// TwinCAT 3 PLC project ExamplePlc
// Company: Sensata Technologies Mechanization
// ProgramVersion: 3.1.4023.0
// libraries:
//   Sensata_Common, * (Sensata Technologies)
//   Sensata_Data, * (Sensata Technologies)
//   Sensata_Device_Comm, * (Sensata Technologies)
//   Sensata_Laser, * (Sensata Technologies)
//   Sensata_Utilities, * (Sensata Technologies)
//   Tc2_Standard, * (Beckhoff Automation GmbH)
//   Tc2_System, * (Beckhoff Automation GmbH)
//   Tc2_Utilities, * (Beckhoff Automation GmbH)
//   Tc3_Module, * (Beckhoff Automation GmbH)
// project tree:
//   0 Program/ GVL_DataTransfer.TcGVL, GVL_HMITags.TcGVL, GVL_LaserMarkingParams.TcGVL, GVL_MESData.TcGVL, GVL_MESData_ActuatorAssembly.TcGVL, GVL_PriorOp.TcGVL, GVL_ProductLimits.TcGVL, GVL_Test.TcGVL, PRG_Main.TcPOU
//   1 Module/0 Machines/ FB_ExampleMachine.TcPOU
//   1 Module/1 Stations/ FB_ExampleStation.TcPOU
//   1 Module/2 Devices/ FB_ExampleDevice.TcPOU
//   / TMethodNames_Cohap.TcDUT, TASK_Main.TcTTO (not stored), TMethod_Controls.TcDUT
// real-time tasks:
//   TASK TASK_Main: cycle T#10ms, priority 20, ADS port 350

// ---- TMethodNames_Cohap.TcDUT
TYPE TMethodNames_Cohap :
STRUCT
	M_init : STRING := 'init';
	M_GetAsicandChannelCardVersion : STRING := 'getSICAndChannelCardVersions';
	M_GetDLLVersion : STRING := 'getDLLVersions';
	M_TestDummy : STRING := 'TestDummy';
	M_TestDummy2 : STRING := 'TestDummy2';
	M_PowerUp : STRING := 'PowerUp';
	M_PowerDown : STRING := 'PowerDown';
	M_readSerialNumber : STRING := 'readSerialNumber';
	M_ReadDeviceOutput : STRING := 'ReadDeviceOutput';
	M_ReadFastChannelData : STRING := 'SENT_readFastChannelData';
	M_initDUT : STRING := 'initDUT';
	M_initialize : STRING := 'initialize';
	
	M_InitLot : STRING := 'InitLot';
//	M_T1Step1 : STRING := '';
//	stM_InitLot	: STRING := 'InitLot';
	stM_t1Precal : STRING := 't1Precal';
	stM_t1Step2 : STRING := 't1Step2';
	stM_t1Step3 : STRING := 't1Step3';
	stM_t2Step1 : STRING := 't2Step1';
	stM_t2Step2 : STRING := 't2Step2';
	stM_t2Step3 : STRING := 't2Step3';	
END_STRUCT
END_TYPE

// ---- TMethod_Controls.TcDUT
TYPE TMethod_Controls :
STRUCT
//		bRunImpMethods_Trigger : BOOL;
//		bRunImpMethods_Result : BOOL;
		bInitializeDeviceComm_Trigger : BOOL;
		bInitializeDeviceComm_Result : BOOL;
		bSetCurrentDevice_Trigger : BOOL;
		bSetCurrentDevice_Result : BOOL;
		M_init_Trigger : BOOL;
        M_init_Result : BOOL;
        M_GetAsicandChannelCardVersion_Trigger : BOOL;
        M_GetAsicandChannelCardVersion_Result : BOOL;
        M_GetDLLVersion_Trigger : BOOL;
        M_GetDLLVersion_Result : BOOL;
        M_TestDummy_Trigger : BOOL;
        M_TestDummy_Result : BOOL;
		M_TestDummy2_Trigger : BOOL;
        M_TestDummy2_Result : BOOL;
        M_PowerUp_Trigger : BOOL;
        M_PowerUp_Result : BOOL;
        M_PowerDown_Trigger : BOOL;
        M_PowerDown_Result : BOOL;
        M_readSerialNumber_Trigger : BOOL;
        M_readSerialNumber_Result : BOOL;
        M_ReadDeviceOutput_Trigger : BOOL;
        M_ReadDeviceOutput_Result : BOOL;
		M_ReadFastChannelData_Trigger : BOOL;
        M_ReadFastChannelData_Result : BOOL;
        M_initDUT_Trigger : BOOL;
        M_initDUT_Result : BOOL;
        M_initialize_Trigger : BOOL;
        M_initialize_Result : BOOL;
		M_initLot_Trigger : BOOL;
		M_initLot_Result : BOOL;
		
		M_t1PreCal_Trigger : BOOL;
		M_t1PreCal_Result : BOOL;
		M_t1Step2_Trigger : BOOL;
		M_t1Step2_Result : BOOL;
		M_t1Step3_Trigger : BOOL;
		M_t1Step3_Result : BOOL;
		M_t2Step1_Trigger : BOOL;
		M_t2Step1_Result : BOOL;
		M_t2Step2_Trigger : BOOL;
		M_t2Step2_Result : BOOL;
		M_t2Step3_Trigger : BOOL;
		M_t2Step3_Result : BOOL;
END_STRUCT
END_TYPE

// ---- 0 Program/GVL_DataTransfer.TcGVL
{attribute 'qualified_only'}
VAR_GLOBAL
//InsertLotHistory
	dintEquipment_Id : DINT;//int
	
	strLot_ID : STRING;//varchar
	strDeviceID :STRING := 'ZSE3230';//varchar
	strAsicType:UDINT := 43;//int
	
//	strTestTime_L1: STRING:='2023/01/27 10:12:11.000';//datetime
//	udintfixture_L1: UDINT:=1;//tinyint
//	bTestStatus_L1 : STRING:='Good';//varchar
//	udintErrorcode_L1 : UDINT:=0;//bigint
//	SerialNumber_L1:UDINT:=180000;//bigint
//	PressureOut_L1:REAL:=1688653;//float
//	TemperatureOut_L1:REAL:=4592369;//float
	
//	bTestStatus_L2 : STRING;//varchar
//	strTestTime_L2: STRING:='2023/01/25 10:12:11.000';//datetime
//	udintErrorcode_L2 : UDINT;
//	udintfixture_L2: UDINT;//tinyint
//	SerialNumber_L2:UDINT;
//	PressureOut_L2:REAL;
//	TemperatureOut_L2:REAL;
//	dintEquipment_Id : DINT;
	
//	strLot_ID : STRING;
//	strDeviceID :STRING;
//	strAsicType:UDINT;//int
	//****************************//
	
	
	strTestTime_L1: STRING;//datetime
	udintfixture_L1: UDINT;//tinyint
	bTestStatus_L1 : STRING:='Good';//varchar
	udintErrorcode_L1 : UDINT:=0;//bigint
	SerialNumber_L1:UDINT;//bigint
	PressureOut_L1:REAL;//float
	TemperatureOut_L1:REAL;//float
	FFTPriorOPstatus_L1: STRING;
	CalT1PriorOPstatus_L1:STRING;
	CalT2PriorOPstatus_L1:STRING;
	ErrorCode_L1:UDINT;
	
	bTestStatus_L2 : STRING;//varchar
	strTestTime_L2: STRING;//datetime
	udintErrorcode_L2 : UDINT;
	udintfixture_L2: UDINT;//tinyint
	SerialNumber_L2:UDINT;
	PressureOut_L2:REAL;
	TemperatureOut_L2:REAL;
	FFTPriorOPstatus_L2: STRING;
	CalT1PriorOPstatus_L2:STRING;
	CalT2PriorOPstatus_L2:STRING;
	ErrorCode_L2:UDINT;//01- prior Op, 02- Invalid SN, 03-Cohap Communication fail
	
	//prior OP 
	
	SerialNumber_temp:UDINT := 989;
	PriorOpTestmode: STRING := 'CalNoBlow';
	PriorOpTestStatus:STRING;
	priorOpResult: STRING;

END_VAR

// ---- 0 Program/GVL_HMITags.TcGVL
{attribute 'qualified_only'}
VAR_GLOBAL
	//machine status 
	//*******
	//Add this line of code to a Program : GVL_HMI.intMachine_State := GVL_Main.fbMachine.P_enumState;
	//*******
	intMachine_State :INT;
	
	// ---------------------------------------------------------------------------
	// Config Screen
	// ---------------------------------------------------------------------------		
	strEngineerPassword: T_MaxString;
	bEngineerAccessAllowed: BOOL;
	strEngineerSetPassword: T_MaxString := 'password';
	bEngineerLogout: BOOL;
	
	//machine overview
	intGood_Parts : INT;
	intBad_Parts : INT;
	intTotal_Parts: INT;
	rYield : REAL;
	dintEquipment_Id : DINT := 191135;
	strSoftware_Rev : STRING := '1.0.0';
	strHMI_Rev : STRING := '1.0';
	bStartBtn : BOOL;
	bStopBtn : BOOL;
	bResetBtn : BOOL;
	bClearBtn : BOOL;
	bUser_Active : BOOL;
	udintPromptMessage : UDINT;
	strUser_Prompt : T_MaxString;
	bLoadDirection: BOOL;
	bDirectionIndicator: BOOL;
	bUserRetryBtn : BOOL;
	bUserAbortBtn : BOOL;
	intStationStatus: INT;
	
	bSetPartIdExternal : BOOL;
	bSetJobIdExternal : BOOL;
	bSetLotIdExternal : BOOL;
	
	strExternalPartId : STRING;
	strExternalJobId : STRING;
	strExternalLotId : STRING;
			
	//Lot Control
	bStart_Lot :BOOL;
	bEnd_Lot : BOOL;
	bLot_Active :BOOL;
	strLot_Num : STRING;
	strJob_Num : STRING;
	strPart_Num : STRING;
	bLimits_Loaded : Bool;
	
	//load unload
	strL1_HCode_Unload : STRING;
	strL2_HCode_Unload : STRING;
	strR1_HCode_Unload : STRING;
	strR2_HCode_Unload : STRING;
	bL1_State_Unload : BOOL;
	bL2_State_Unload : BOOL;
	bR1_State_Unload : BOOL;
	bR2_State_Unload : BOOL;
	
	//conditioner
	intNum_Cycles : INT;
	intOn_Time : INT;
	intOff_Time : INT;
	intCycles_Run :INT;
	bL1_Cond_State : BOOL;
	bL2_Cond_State : BOOL;
	bR1_Cond_State : BOOL;
	bR2_Cond_State : BOOL;
	strL1_Cond_HCode : STRING;
	strL2_Cond_HCode : STRING;
	strR1_Cond_HCode : STRING;
	strR2_Cond_HCode : STRING;
		
	//contact resistance	
	strCR_L1_HCode : STRING;
	rCR_L1_CR : REAL;
	rCR_L1_M1R : REAL;
	rCR_L1_M1V : REAL;
	rCR_L1_M1C : REAL;
	rCR_L1_M2R : REAL;
	rCR_L1_M2V : REAL;
	rCR_L1_M2C : REAL;
	rCR_L1_A1R : REAL;
	rCR_L1_A1V : REAL;
	rCR_L1_A1C : REAL;
	rCR_L1_A2R : REAL;
	rCR_L1_A2V : REAL;
	rCR_L1_A2C : REAL;
	bL1_CR_State : BOOL;
	
	strCR_L2_HCode : STRING;
	rCR_L2_CR : REAL;
	rCR_L2_M1R : REAL;
	rCR_L2_M1V : REAL;
	rCR_L2_M1C : REAL;
	rCR_L2_M2R : REAL;
	rCR_L2_M2V : REAL;
	rCR_L2_M2C : REAL;
	rCR_L2_A1R : REAL;
	rCR_L2_A1V : REAL;
	rCR_L2_A1C : REAL;
	rCR_L2_A2R : REAL;
	rCR_L2_A2V : REAL;
	rCR_L2_A2C : REAL;
	bL2_CR_State : BOOL;
	
	strCR_R1_HCode : STRING;
	rCR_R1_CR : REAL;
	rCR_R1_M1R : REAL;
	rCR_R1_M1V : REAL;
	rCR_R1_M1C : REAL;
	rCR_R1_M2R : REAL;
	rCR_R1_M2V : REAL;
	rCR_R1_M2C : REAL;
	rCR_R1_A1R : REAL;
	rCR_R1_A1V : REAL;
	rCR_R1_A1C : REAL;
	rCR_R1_A2R : REAL;
	rCR_R1_A2V : REAL;
	rCR_R1_A2C : REAL;	
	bR1_CR_State : BOOL;
	
	strCR_R2_HCode : STRING;
	rCR_R2_CR : REAL;
	rCR_R2_M1R : REAL;
	rCR_R2_M1V : REAL;
	rCR_R2_M1C : REAL;
	rCR_R2_M2R : REAL;
	rCR_R2_M2V : REAL;
	rCR_R2_M2C : REAL;
	rCR_R2_A1R : REAL;
	rCR_R2_A1V : REAL;
	rCR_R2_A1C : REAL;
	rCR_R2_A2R : REAL;
	rCR_R2_A2V : REAL;
	rCR_R2_A2C : REAL;
	bR2_CR_State : BOOL;
		
	//hipot	
	strHp_L1_HCode : STRING;
	strHp_L2_HCode : STRING;
	strHp_R1_HCode : STRING;
	strHp_R2_HCode : STRING;
	//to be deleted
	bL1_Hp_State : BOOL;
	bL2_Hp_State : BOOL;
	bR1_Hp_State : BOOL;	
	bR2_Hp_State : BOOL;
	
	rHp_FT_L1 : REAL;
	rHp_FT_L2 : REAL;
	rHp_FT_R1 : REAL;
	rHp_FT_R2 : REAL;

	rHp_Res_L1 : REAL;
	rHp_Res_L2 : REAL;
	rHp_Res_R1 : REAL;
	rHp_Res_R2 : REAL;
	
	strHp_Msg_L1 : STRING;
	strHp_Msg_L2 : STRING;
	strHp_Msg_R1 : STRING;
	strHp_Msg_R2 : STRING;
	
	HP_testName : STRING;
	//not used on HMI
	rHp_BDC_L1 : REAL;
	rHp_ARC_L1 : REAL;
	rHp_Result_L1 : REAL;
	rHp_BDC_L2 : REAL;
	rHp_ARC_L2 : REAL;
	rHp_Result_L2 : REAL;
	rHp_BDC_R1 : REAL;
	rHp_ARC_R1 : REAL;
	rHp_Result_R1 : REAL;
	rHp_BDC_R2 : REAL;
	rHp_ARC_R2 : REAL;
	rHp_Result_R2 : REAL;
	//AB proposed new Tags
	strNestAErrorMsg:STRING;
	strNestBErrorMsg:STRING;
	strNestCErrorMsg:STRING;
	strNestDErrorMsg:STRING;
	
	rHPMeasured_MML1:REAL;
	rHPMeasured_MML2:REAL;
	rHPMeasured_MMR1:REAL;
	rHPMeasured_MMR2:REAL;
	
	rHPMeasured_MMIRL1:REAL;
	rHPMeasured_MMIRL2:REAL;
	rHPMeasured_MMIRR1:REAL;
	rHPMeasured_MMIRR2:REAL;
	
	rHPMeasured_AAL1:REAL;
	rHPMeasured_AAL2:REAL;
	rHPMeasured_AAR1:REAL;
	rHPMeasured_AAR2:REAL;
	
	rHPMeasured_AuxIRL1:REAL;
	rHPMeasured_AuxIRL2:REAL;
	rHPMeasured_AuxIRR1:REAL;
	rHPMeasured_AuxIRR2:REAL;
	
	rHPMeasured_MainCoilopenL1:REAL;
	rHPMeasured_MainCoilopenL2:REAL;
	rHPMeasured_MainCoilopenR1:REAL;
	rHPMeasured_MainCoilopenR2:REAL;
	
	rHPMeasured_MainCoilIRL1:REAL;
	rHPMeasured_MainCoilIRL2:REAL;
	rHPMeasured_MainCoilIRR1:REAL;
	rHPMeasured_MainCoilIRR2:REAL;
	
	rHPMeasured_MainCoilClosedL1:REAL;
	rHPMeasured_MainCoilClosedL2:REAL;
	rHPMeasured_MainCoilClosedR1:REAL;
	rHPMeasured_MainCoilClosedR2:REAL;
	
	
	//PUV_DOV
	strPUV_L1_HCode : STRING;
	strPUV_L2_HCode : STRING;
	strPUV_R1_HCode : STRING;
	strPUV_R2_HCode : STRING;
	
	bL1_puv_State : BOOL;
	bL2_puv_State : BOOL;
	bR1_puv_State : BOOL;
	bR2_puv_State : BOOL;
	
	rPuv_L1 : REAL;
	rDov_L1 : REAL;	
	rPuc_L1 : REAL;
	rDoc_L1 : REAL;
	rPuv_L2 : REAL;
	rDov_L2 : REAL;	
	rPuc_L2 : REAL;
	rDoc_L2 : REAL;
	rPuv_R1 : REAL;
	rDov_R1 : REAL;	
	rPuc_R1 : REAL;
	rDoc_R1 : REAL;
	rPuv_R2 : REAL;
	rDov_R2 : REAL;	
	rPuc_R2 : REAL;
	rDoc_R2 : REAL;
	
	arrCoilPUV: ARRAY[1..4] OF LREAL;
	arrCoilDOV: ARRAY[1..4] OF LREAL;
	arrCoilResistance: ARRAY[1..4] OF LREAL;
		
	//functional test	
	strFT_L1_HCode : STRING;
	strFT_L2_HCode : STRING;
	strFT_R1_HCode : STRING;
	strFT_R2_HCode : STRING;
	
	bL1_ft_State : BOOL;
	bL2_ft_State : BOOL;
	bR1_ft_State : BOOL;
	bR2_ft_State : BOOL;
	
	MainOperatTime_L1 : REAL;
	MainReleaseTime_L1 : REAL;	
	AuxOperateTime_L1 : REAL;
	AuxReleaseTime_L1 : REAL;
	RSim_L1 : REAL;
	MainOperatTime_L2 : REAL;
	MainReleaseTime_L2 : REAL;	
	AuxOperateTime_L2 : REAL;
	AuxReleaseTime_L2 : REAL;
	RSim_L2 : REAL;
	MainOperatTime_R1 : REAL;
	MainReleaseTime_R1 : REAL;	
	AuxOperateTime_R1 : REAL;
	AuxReleaseTime_R1 : REAL;
	RSim_R1 : REAL;
	MainOperatTime_R2 : REAL;
	MainReleaseTime_R2 : REAL;	
	AuxOperateTime_R2 : REAL;
	AuxReleaseTime_R2 : REAL;
	RSim_R2 : REAL;
	
	//laser mark	
	bLaser_Connected_State : BOOL;
	bLaser_Mark_Status : BOOL;
	bLaser_Mark_Status_L1 : BOOL; //Marking Status of Part in Nest L1
	bLaser_Mark_Status_L2 : BOOL; //Marking Status of Part in Nest L2
	bLaser_Mark_Status_R1 : BOOL; //Marking Status of Part in Nest R1
	bLaser_Mark_Status_R2 : BOOL; //Marking Status of Part in Nest R2
	
	//Station PBs
	bDialTableRetry: BOOL;
	bDialTableAbort: BOOL;
	bCondRetry : BOOL;
	bCondAbort : BOOL;
	bCRRetry : BOOL;
	bCRAbort : BOOL;
	bHPRetry : BOOL;
	bHPAbort : BOOL;
	bPUVRetry : BOOL;
	bPUVAbort : BOOL;
	bFTRetry : BOOL;
	bFTAbort : BOOL;
	bLaserRetry: BOOL;
	bLaserAbort: BOOL;
	
	//Station Messages
	strLoadUserMsg : T_MaxString;
	strCondUserMsg : T_MaxString;
	strCRUserMsg : T_MaxString;
	strHPUserMsg : T_MaxString;
	strPUVUserMsg : T_MaxString;
	strFTUserMsg : T_MaxString;
	
	//Disable stations from HMI
	bDisableDialTable : BOOL;
	bDisableLoadUnload : BOOL;
	bDisableConditioner : BOOL;
	bDisableCR : BOOL;
	bDisableHiPot : BOOL;
	bDisableLaserMark : BOOL;
	bDisablePUVDOV : BOOL;
	bDisableFunctionTest : BOOL;	
	
	udintDialTablePrompt: UDINT;
	udintLoadUnloadPrompt: UDINT;
	udintConditionerPrompt: UDINT;
	udintContactResistancePrompt: UDINT;
	udintHiPotPrompt: UDINT;
	udintLaserPrompt: UDINT;
	udintPUVDOVPrompt: UDINT;
	udintFunctionTestPrompt: UDINT;
	
	bDialTablePromptActive: BOOL;
	bLoadUnloadPromptActive: BOOL;
	bConditionerPromptActive: BOOL;
	bContactResistancePromptActive: BOOL;
	bHiPotPromptActive: BOOL;
	bLaserPromptActive: BOOL;
	bPUVDOVPromptActive: BOOL;
	bFunctionTestPromptActive: BOOL;
	
	udintDialTableFault: UDINT;
	udintLoadUnloadFault: UDINT;
	udintConditionerFault: UDINT;
	udintContactResistanceFault: UDINT;
	udintHiPotFault: UDINT;
	udintLaserFault: UDINT;
	udintPUVDOVFault: UDINT;
	udintFunctionTestFault: UDINT;
	
	bDialTableFaulted: BOOL;
	bLoadUnloadFaulted: BOOL;
	bConditionerFaulted: BOOL;
	bContactResistanceFaulted: BOOL;
	bHiPotFaulted: BOOL;
	bLaserFaulted: BOOL;
	bPUVDOVFaulted: BOOL;
	bFunctionTestFaulted: BOOL;

	
	intDialTableState: INT;
	intLoadUnloadState: INT;
	intConditionerState: INT;
	intContactResistanceState: INT;
	intHiPotState: INT;
	intLaserState: INT;
	intPUVDOVState: INT;
	intFunctionTestState: INT;
	
	//Station and Nest failed consecutively 3 times
	//intStationNumFailed: INT;
	//intNestNumFailed: INT;
	arrStationNestNumFailed: ARRAY[1..2] OF INT;
	
	//IO Screen
	arrDigitalInputs: ARRAY[1..32] OF BOOL;
	arrRemoteInputs: ARRAY[1..48] OF BOOL;
	arrIOLinkInputs: ARRAY[1..4] OF BOOL;
	arrDigitalOutputStatus: ARRAY[1..120] OF BOOL;
	arrRelayOutputStatus: ARRAY[1..4] OF BOOL;
	arrPneumaticOutputStatus: ARRAY[1..32] OF BOOL;
	arrGuardDoors: ARRAY[1..16] OF BOOL;
//	arrMultiTimestampInputs: ARRAY[1..8] OF ST_EL1258_Inputs_Channel;
	
END_VAR

// ---- 0 Program/GVL_LaserMarkingParams.TcGVL
{attribute 'qualified_only'}
VAR_GLOBAL
	strHousingCode_L1 : STRING;	

	strCustomerDeviceID_L1 : STRING;
	strBlock0_L1 : STRING;
	strBlock1_L1 : STRING;
	strBlock2_L1 : STRING;
	strBlock3_L1 : STRING;
	strBlock4_L1 : STRING;
	strBlock5_L1 : STRING;
	strBlock6_L1 : STRING;
	strBlock7_L1 : STRING;
	strBlock8_L1 : STRING;
	strBlock9_L1 : STRING;
	strBlock10_L1 : STRING;
	
	strHousingCode_L2 : STRING;	
	
	strCustomerDeviceID_L2 : STRING;
	strBlock0_L2 : STRING;
	strBlock1_L2 : STRING;
	strBlock2_L2 : STRING;
	strBlock3_L2 : STRING;
	strBlock4_L2 : STRING;
	strBlock5_L2 : STRING;
	strBlock6_L2 : STRING;
	strBlock7_L2 : STRING;
	strBlock8_L2 : STRING;
	strBlock9_L2  : STRING;
	strBlock10_L2 : STRING;

	strHousingCode_R1 : STRING;	
	
	strCustomerDeviceID_R1 : STRING;
	strBlock0_R1 : STRING;
	strBlock1_R1 : STRING;
	strBlock2_R1 : STRING;
	strBlock3_R1 : STRING;
	strBlock4_R1 : STRING;
	strBlock5_R1 : STRING;
	strBlock6_R1 : STRING;
	strBlock7_R1 : STRING;
	strBlock8_R1 : STRING;
	strBlock9_R1 : STRING;
	strBlock10_R1 : STRING;
	
	strHousingCode_R2 : STRING;	
	
	strCustomerDeviceID_R2 : STRING;
	strBlock0_R2 : STRING;
	strBlock1_R2 : STRING;
	strBlock2_R2 : STRING;
	strBlock3_R2 : STRING;
	strBlock4_R2 : STRING;
	strBlock5_R2 : STRING;
	strBlock6_R2 : STRING;
	strBlock7_R2 : STRING;
	strBlock8_R2 : STRING;
	strBlock9_R2 : STRING;
	strBlock10_R2 : STRING;
	
END_VAR

// ---- 0 Program/GVL_MESData.TcGVL
{attribute 'qualified_only'}
VAR_GLOBAL
	//Lot Information
	LotBarcode : STRING;// := '80600600+57805702+23330166A+200';
	
	LotNo : STRING;
	ProductNo : STRING;
	OrderNo : STRING;
	Quantity : INT;
	OperatorID : STRING;
	ShiftLeader : STRING;
	MachineID : STRING;
	LotIdent : INT;
	PiecesLeft : INT;
	PiecesOK : INT;
	PiecesNOK : INT;
	LotInfoResponseMessages : ARRAY[1..100] OF STRING;
	
	//Operator Information 1
	OperatorBarcode : STRING;
	OperatorInfoResponse : STRING;	
	OperatorInfoResponseMessages : ARRAY[1..100] OF STRING;
	
	//Start Lot Information 1
	StartLotResponse : STRING;
	StartLotResponseMessages : ARRAY[1..100] OF STRING;
	
	//Prod Lot Components 1, 2 , 3
	Comp1_ident: LINT;          // Equivalent to private long ident;
   	Comp1_ident2: INT;          // Equivalent to private int ident2;
    Comp1_seria: STRING;        // Equivalent to private string seria;
    Comp1_quan: INT;            // Equivalent to private int quan;
    Comp1_result: INT;        // Equivalent to private short result;
    Comp1_resultText: STRING;   // Equivalent to private string resultText;
    Comp1_actualQuan: INT;      // Equivalent to private int actualQuan;
    Comp1_item: STRING;         // Equivalent to private string item;
	
	Comp2_ident: LINT;          // Equivalent to private long ident;
   	Comp2_ident2: INT;          // Equivalent to private int ident2;
    Comp2_seria: STRING;        // Equivalent to private string seria;
    Comp2_quan: INT;            // Equivalent to private int quan;
    Comp2_result: INT;        // Equivalent to private short result;
    Comp2_resultText: STRING;   // Equivalent to private string resultText;
    Comp2_actualQuan: INT;      // Equivalent to private int actualQuan;
    Comp2_item: STRING;         // Equivalent to private string item;
	
	Comp3_ident: LINT;          // Equivalent to private long ident;
   	Comp3_ident2: INT;          // Equivalent to private int ident2;
    Comp3_seria: STRING;        // Equivalent to private string seria;
    Comp3_quan: INT;            // Equivalent to private int quan;
    Comp3_result: INT;        // Equivalent to private short result;
    Comp3_resultText: STRING;   // Equivalent to private string resultText;
    Comp3_actualQuan: INT;      // Equivalent to private int actualQuan;
    Comp3_item: STRING;         // Equivalent to private string item;
	
	//ComponentsValidation 1, 2, 3
	ComponentValidation1Response : BOOL;
	ComponentValidation2Response : BOOL;
	ComponentValidation3Response : BOOL;
	
	//Get Machine Settings 1
	MachineSettingStructure : STRING;
	in_MachSetResult : BOOL;
	in_MachSetStructResponse : T_MaxString;
	
	//AddScrapCompByReason1
	
	//ScrapInfo
	ScrapCode : INT;
	ScrapCount : INT;
	ScrapCodeDescr : STRING;
	
	//Response 
	AddScrapComponentByReasonResponse : BOOL;
	
	//EndComponentLot1
	UsedComponentQuantity : INT;
	ComponentLotFinished : BOOL;
	//Response 
	EndLotComponentResponse : BOOL;
	
	
	//GetMachineDefects
	GetMachineDefects1Success : BOOL;
	Scrap1_ScrapCode : INT;
	Scrap1_ScrapCount : INT;
	Scrap1_ScrapCodeDescr : STRING;	
	
	//AddMESMachineEvent
	MESMachineID : STRING;
	MESStationID : INT;
	MESEventCode : STRING;
	MESEventMessage : STRING;
	MESEventType : INT;
	MESEventOperatorID : STRING;
	
	MESResponseEventID : LINT;
	
	//UpdateMESMachineEvent
	MESIsResolvedStatus : BOOL;
	MESResolutionNotes : STRING;
	MESDateTimeResolved : DATE;
	MESUpdateEventID : LINT;
	
END_VAR

// ---- 0 Program/GVL_MESData_ActuatorAssembly.TcGVL
{attribute 'qualified_only'}
VAR_GLOBAL
	//Lot Information
	LotBarcode : STRING;// := '80600600+57805702+23330166A+200';
	
	LotNo : STRING;
	ProductNo : STRING;
	OrderNo : STRING;
	Quantity : INT;
	OperatorID : STRING;
	ShiftLeader : STRING;
	MachineID : STRING;
	LotIdent : INT;
	PiecesLeft : INT;
	PiecesOK : INT;
	PiecesNOK : INT;
	LotInfoResponseMessages : ARRAY[1..100] OF STRING;
	
	//Operator Information 1
	OperatorBarcode : STRING;
	OperatorInfoResponse : STRING;	
	OperatorInfoResponseMessages : ARRAY[1..100] OF STRING;
	
	//machine settings
	
	//Start Lot Information 1
	StartLotResponse : STRING;
	StartLotResponseMessages : ARRAY[1..100] OF STRING;
	
	//Prod Lot Components 1, 2 , 3
	Comp1_ident: LINT;          // Equivalent to private long ident;
   	Comp1_ident2: INT;          // Equivalent to private int ident2;
    Comp1_seria: STRING;        // Equivalent to private string seria;
    Comp1_quan: INT;            // Equivalent to private int quan;
    Comp1_result: INT;        // Equivalent to private short result;
    Comp1_resultText: STRING;   // Equivalent to private string resultText;
    Comp1_actualQuan: INT;      // Equivalent to private int actualQuan;
    Comp1_item: STRING;         // Equivalent to private string item;
	
	Comp2_ident: LINT;          // Equivalent to private long ident;
   	Comp2_ident2: INT;          // Equivalent to private int ident2;
    Comp2_seria: STRING;        // Equivalent to private string seria;
    Comp2_quan: INT;            // Equivalent to private int quan;
    Comp2_result: INT;        // Equivalent to private short result;
    Comp2_resultText: STRING;   // Equivalent to private string resultText;
    Comp2_actualQuan: INT;      // Equivalent to private int actualQuan;
    Comp2_item: STRING;         // Equivalent to private string item;
	
	Comp3_ident: LINT;          // Equivalent to private long ident;
   	Comp3_ident2: INT;          // Equivalent to private int ident2;
    Comp3_seria: STRING;        // Equivalent to private string seria;
    Comp3_quan: INT;            // Equivalent to private int quan;
    Comp3_result: INT;        // Equivalent to private short result;
    Comp3_resultText: STRING;   // Equivalent to private string resultText;
    Comp3_actualQuan: INT;      // Equivalent to private int actualQuan;
    Comp3_item: STRING;         // Equivalent to private string item;
	
	//ComponentsValidation 1, 2, 3
	ComponentValidation1Response : BOOL;
	ComponentValidation2Response : BOOL;
	ComponentValidation3Response : BOOL;
	
	//Get Machine Settings 1
	MachineSettingStructure : STRING;
	in_MachSetResult : BOOL;
	in_MachSetStructResponse : T_MaxString;
	
	//AddScrapCompByReason1
	
	//ScrapInfo
	ScrapCode : INT;
	ScrapCount : INT;
	ScrapCodeDescr : STRING;
	
	//Response 
	AddScrapComponentByReasonResponse : BOOL;
	
	//EndComponentLot1
	UsedComponentQuantity : INT;
	ComponentLotFinished : BOOL;
	//Response 
	EndLotComponentResponse : BOOL;
	
	
	//GetMachineDefects
	GetMachineDefects1Success : BOOL;
	Scrap1_ScrapCode : INT;
	Scrap1_ScrapCount : INT;
	Scrap1_ScrapCodeDescr : STRING;	
	
	//AddMESMachineEvent
	MESMachineID : STRING;
	MESStationID : INT;
	MESEventCode : STRING;
	MESEventMessage : STRING;
	MESEventType : INT;
	MESEventOperatorID : STRING;
	
	MESResponseEventID : LINT;
	
	//UpdateMESMachineEvent
	MESIsResolvedStatus : BOOL;
	MESResolutionNotes : STRING;
	MESDateTimeResolved : DATE;
	MESUpdateEventID : LINT;
	
	
	
END_VAR

// ---- 0 Program/GVL_PriorOp.TcGVL
{attribute 'qualified_only'}
VAR_GLOBAL
	strHousingCode_L1 : STRING;
	bLaserMarked_L1 : BOOL;
END_VAR

// ---- 0 Program/GVL_ProductLimits.TcGVL
{attribute 'qualified_only'}
VAR_GLOBAL
	strPart_Num : STRING := 'GV354-006'; // := 'GXV600-009';
	strToolingBarcodeRequired : STRING;
	intBarcodeLocation : INT;
	
	
	//Conditioner Station
	bEnableConditioner : BOOL;
	intNumberOfCyclesToRun : INT := 500;
	intOperateTime : INT := 8;
	intReleaseTime : INT := 18;
	
	//CR Station
	bEnableCR : BOOL;
	bAuxPresent : BOOL;
	bEnableDipTest : BOOL;
	bEnableEMFTest : BOOL;
	bEndTestInRange : BOOL;
	intInitialWaitTime : INT;
	intMaxTestPulseTime : INT;
	intNumberofContResToCheck : INT;
	intNumberofPulses : INT;//Currently for rivian only
	intPulseOFFTime : INT;
	lrealInAuxResistanceMin : LREAL; 
	lrealInAuxResistanceMax : LREAL;
	lrealInCoilResistanceMin : LREAL; 
	lrealInCoilResistanceMax : LREAL; 
	lrealInMainsResistanceMin : LREAL;
	lrealInMainsResistanceMax : LREAL;
	lrealInMainsResistanceRangeMax : LREAL;
	lrealInMainsResistanceLastPointMax : LREAL;	
	lrealSetCurrentCoil : LREAL;
	lrealSetVoltageCoil : LREAL;
	lrealSetCloseTestCurrentMain : LREAL;
	lrealSetCloseTestVoltageMain : LREAL;
	lrealSetTestingCurrentMain : LREAL;
	lrealSetTestingVoltageMain : LREAL;
	lrealMainsCurrentErrorPct : LREAL;

	bEnableHP:BOOL;
	bDBParamsAux2APresent:BOOL:=TRUE;
	bDBParamsAux2BPresent:BOOL;
	udintEquipmentCountCycle:UDINT;
	lrealTestVoltageHP:LREAL;
	lrealDwellTime:LREAL;
	lrealRampTime:LREAL;
	lrealMinCurrentHP:LREAL;
	lrealMaxCurrentHP:LREAL;
	lrealTestVoltageIR:LREAL;
	lrealMinResistanceIR:LREAL;
	lrealMaxResistanceIR:LREAL;
	strDUT_HP:STRING;
	
	//TestVoltage for Aux test
	lrTestVoltageAuxHP: LREAL;
	//DwellTime for Aux-Aux HP test
	lrTestDwellTimeAuxHP:LREAL;
	//RampTime for Aux-Aux HP test
	lrTestRampTimeAuxHP :LREAL;
	//MinAcceptable current for Aux-Aux HP test
	lrMinCurrentAuxHP :LREAL;
	//MaxAcceptable current for Aux-Aux HP test
	lrMaxCurrentAuxHP :LREAL;
	
	//PUVDOV Station
	bEnablePUV:BOOL;
	bBinarySearchEnabled: BOOL; 	
	bVoltageTest: BOOL;        	
	udintBinarySearchPoints : UDINT;	
	timeContactCloseCheck : UINT; 	
	timePowerFailCheck: UINT;
	timePowerSupplyStabilize: UINT;	
	lrealDefaultErrValue : LREAL;
	lrealPickUpUSLVoltage: LREAL;	
	lrealPickUpLSLVoltage: LREAL; 
	lrealPickUpBufferVoltage: LREAL;
	lrealPickUpUSLCurrent: LREAL;
	lrealPickUpLSLCurrent: LREAL;
	lrealPickUpBufferCurrent: LREAL;
	lrealCoilNominalVoltage: LREAL; 
	lrealCoilNominalCurrent: LREAL;
	lrealDropOutUSLVoltage: LREAL; 
	lrealDropOutLSLVoltage: LREAL;
	lrealDropOutBufferVoltage: LREAL;	
	lrealDropOutUSLCurrent: LREAL;	
	lrealDropOutLSLCurrent: LREAL;
	lrealDropOutBufferCurrent: LREAL;
	lrealMaxCurrentSet: LREAL;
	lrealMaxVoltageSet: LREAL;
	
	//Laser Station
	bEnableLaser:BOOL;
	strLaserBlock_0:STRING;
	strLaserBlock_1:STRING;
	strLaserBlock_2:STRING;
	strLaserBlock_3:STRING;
	strLaserBlock_4:STRING;
	strLaserBlock_5:STRING;
	strLaserBlock_6:STRING;
	strLaserBlock_7:STRING;
	strLaserBlock_8:STRING;
	strLaserBlock_9:STRING;
	strLaserBlock_10:STRING;
	
	//FT Station
	bEnableFT:BOOL;
	realMainsOTMin : REAL;
	realMainsOTMax : REAL;
	realAuxOTMin : REAL;
	realAuxOTMax : REAL;
	realMainsRTMin : REAL;
	realMainsRTMax : REAL;
	realAuxRTMin : REAL;
	realAuxRTMax : REAL;
	realRSimMin :REAL;
	realRSimMax:REAL;
	
	//Tooling Barcode
	strExpectedToolingBarcode: Tc2_System.T_MaxString;//Remove after db update 
	
	//Pallet Barcode
	strExpectedPalletBarcode : Tc2_System.T_MaxString;
END_VAR

// ---- 0 Program/GVL_Test.TcGVL
{attribute 'qualified_only'}
VAR_GLOBAL
	temperature : REAL;
	Pressure : REAL;
	
	startCommand : BOOL;
	stopCommand : BOOL;
	
END_VAR

// ---- 0 Program/PRG_Main.TcPOU
PROGRAM PRG_Main
VAR
	bTestInput: BOOL;
	bTestOutput: BOOL;
	fbMachine: FB_ExampleMachine;
	fbStation1: FB_ExampleStation;
	fbStation2: FB_ExampleStation;
	fbStation3: FB_ExampleStation;
	fbStation4: FB_ExampleStation;
	bStart: BOOL;
	bAbort: BOOL;
	bReset: BOOL;
	bStop: BOOL;
	bSuspend: BOOL;
	fbDevice1: FB_ExampleDevice;
	fbDevice2: FB_ExampleDevice;
	fbDevice3: FB_ExampleDevice;
	fbDevice4: FB_ExampleDevice;
	bPoweredOn: BOOL;
//	FB_AdsDeviceAPI_0: FB_AdsDeviceAPI;
	FB_AdsDeviceAPI_0 : FB_AdsCommandRouter;
//	FB_AdsDeviceAPI_1 : FB_AdsCommandRouter;
	MyLaser1: FB_KeyenceLaserMarkerMDX2000;
	(* Database handler FB. *)
//	in_fbDataHandler: REFERENCE TO FB_Data;

///////////////////////////////////////////////////////////////////////////
///////////////Laser Marking Testing////////////////////////////////////
///////////////////////////////////////////////////////////////////////////


	bConnectToLaserMarker: BOOL;
	bRes_LaserConnected: BOOL;
	
	bTestADSServer: BOOL;
	strTarget: T_MaxString;
	strCommand: T_MaxString;
	arrParams: T_ApiMethodParameters;
	MyResults: T_MaxString;
	bInterfaceTest : BOOL;
	temp: BOOL;
	
	
	bDisconnectFromLaserMarker: BOOL;
	bRes_LaserDisconnected: BOOL;
	
	bPeakCurrentProgramInLaser: BOOL;
	bRes_PeakCurrentProgramInLaser: BOOL;
	
	bSendProgramToLaser: BOOL;
	bRes_SendProgramtoLaser: BOOL;
	filepath : STRING;
	LaserMemoryLocation : INT;
	
	bSaveCurrentLaserProgramtoPC : BOOL;
	bRes_SaveCurrentLaserProgramtoPC: BOOL;
	LaserProgramFolderPath: STRING;
	
	bGetCurrentProgram : BOOL;
	bRes_GetCurrentProgram : BOOL;
	CurrentProgramName : T_MaxString;
	
	bStartMarking: BOOL;
	bRes_StartMarking: BOOL;
	
	bStopMarking: BOOL;
	bRes_StopMarking: BOOL;
	
	bClearLaserErrors: BOOL;
	bRes_ClearLaserErrors: BOOL;
	
	bUpdateProgramBlockInTheLaser: BOOL;
	bRes_UpdateProgramBlockInTheLaser: BOOL;
	_blockNumber: INT;
	_blockData: STRING;
	_blockType : BlockTypes;
	
	bGetLaserStatus: BOOL;
	bRes_GetLaserStatus: BOOL;
	_string_laserstatus : STRING;
	
	bGetLaserErrorStatus: BOOL;
	bRes_GetLaserErrorStatus: BOOL;
	_bIsLaserError : BOOL;
	
	bGetLaserActivatedStatus: BOOL;
	bRes_GetLaserActivatedStatus: BOOL;
	_bIsLaserActivated : BOOL;
	
	bGetLaserMarkingStatus: BOOL;
	bRes_GetLaserMarkingStatus: BOOL;
	_bIsLaserMarking : BOOL;
	
	bRes_Reset: BOOL;
	bResetErrors: BOOL;
	
	bUpdateProgramBlockMarkEnabledInTheLaser: BOOL;
	bRes_UpdateProgramBlockMarkEnabledInTheLaser: BOOL;
	_bool_markenabled : BOOL;
	_blockType_enum : BlockTypes;
	
	UpdateSingleBlockMarkEnabledIntheLaser_Success: BOOL;
	_bUpdateSingleBlockDataSuccess : BOOL;
	_bUpdateSingleBlockMarkEnabled_Success : BOOL;
	
	bUpdateAllMarkingInfo: BOOL;
	LastBlockToMark : INT;
	_OneTimeArrayBuild : BOOL := TRUE;
	BlockInfoArray : ARRAY [0..255] OF OneBlockInfo;
	bRes_UpdateAllMarkingInfo: BOOL;
	
	
	intIndex: INT;
	intIndex2 : INT;
	inst_intStep: INT := 0;
	_tempString : STRING;
	
	bRes_UpdateAllMarkInfo : ARRAY [0..255] OF BOOL;
	bUpdateAllMarkingInfo_MethodCall: BOOL;
	bRes_UpdateAllMarkingInfo_MethodCall: BOOL;
	
	
	fbDataHandler: FB_DataTracker;
	fbDataHandler2: FB_DataTracker;
	fbDatabaseCommandRouter: FB_AdsCommandRouter;
	_inst_bDataTransferred: BOOL;
	
	// (* Name of the parameters database transfer ID. *)
	in_strParametersDatabaseName: T_MaxString := 'GetLimits';
	in_strParametersDBNameLaserLimits_L1 : T_MaxString := 'GetLaserMarkingParams_L1';
	in_strParametersDBNameLaserLimits_L2 : T_MaxString := 'GetLaserMarkingParams_L2';
	in_strParametersDBNameLaserLimits_R1 : T_MaxString := 'GetLaserMarkingParams_R1';
	in_strParametersDBNameLaserLimits_R2 : T_MaxString := 'GetLaserMarkingParams_R2';	
	_inst_bLaserLimitsDataTransferred_L1 : BOOL;
	_inst_bLaserLimitsDataTransferred_L2 : BOOL;
	_inst_bLaserLimitsDataTransferred_R1 : BOOL;
	_inst_bLaserLimitsDataTransferred_R2 : BOOL;
	
	bGetLimitsFromDB : BOOL;
	
	bGetLaserParamsFromDB_L1 : BOOL;
	bGetLaserParamsFromDB_L2 : BOOL;
	bGetLaserParamsFromDB_R1 : BOOL;
	bGetLaserParamsFromDB_R2 : BOOL;
	
	bPerformPriorOp_Smart: BOOL;
	in_strParametersDBName_SmartWater : T_MaxString := 'GetPriorOPA';
	_inst_bPriorOp_Smart: BOOL;
	
	bPerformPriorOp_FFT: BOOL;
	in_strParametersDBName_FFTLaser_L1 : T_MaxString := 'LaserMarkCheckL1';
	_inst_bPriorOp_FFT: BOOL;
	
	Temp_CR_LOOKUP_NestL1 : INT;
	iLengthDataMatrixNestL1 : INT;
	ParamsArrayNestA : STRING;
	
///////////////////////////////////////////////////////////////////////////
///////////////MES Data Tracking Testing////////////////////////////////////
///////////////////////////////////////////////////////////////////////////

	
	fbDataHandler3: FB_MESDataTracking;
	bPerformGetLotInfoFromLotBarcode: BOOL;
	_inst_bGetLotInfo_LotBarcode: BOOL;
	in_strParamDBName_GetLotInfo: T_MaxString := 'GetLotInfo1';
	
	bPerformGetOpInfoFromOpBarcode: BOOL;
	in_strParamDBName_GetOpInfo: T_MaxString := 'GetOperatorInfo1';
	_inst_bGetOpInfo_OpBarcode: BOOL;
	
	bPerformStartLot : BOOL;
	_inst_bStartLot : BOOL;
	in_strParamDBName_StartLot : T_MaxString := 'StartLot1';
	
	bPerformGetProdLotComponents : BOOL;
	_inst_bGetProdLotComponents : BOOL;
	in_strParamDBName_GetProdLotComps : T_MaxString := 'GetProdLotComponents1';
	
	bPerformComponentValidation1 : BOOL;
	_inst_bCompValidation1 : BOOL;
	in_strParamDBName_Comp1Validation1 : T_MaxString := 'ComponentValidation1';
	
	bPerformComponentValidation2 : BOOL;
	_inst_bCompValidation2 : BOOL;
	in_strParamDBName_Comp1Validation2 : T_MaxString := 'ComponentValidation2';
	
	bPerformComponentValidation3 : BOOL;
	_inst_bCompValidation3 : BOOL;
	in_strParamDBName_Comp1Validation3 : T_MaxString := 'ComponentValidation3';
	
	bPerformGetMachineSettings : BOOL;
	_inst_bGetMachineSettings : BOOL;
	in_strParamDBName_GetMachSetting : T_MaxString := 'GetMachineSettings1';
	
	bPerformAddScrapCompByReason : BOOL;
	_inst_bAddScrapCompByReason : BOOL;
	in_strParamDBName_AddScrapCompByReason : T_MaxString := 'AddScrapComponentByReason1';
	
	bPerformEndLotComp : BOOL;
	_inst_bEndLotComp : BOOL;
	in_strParamDBName_EndLotComp : T_MaxString := 'EndLotComponent1';
	
	bPerformGetMachineDefects : BOOL;
	_inst_bGetMachineDefects : BOOL;
	in_strParamDBName_GetMachDefects : T_MaxString := 'GetMachineDefects1';

	
///////////////////////////////////////////////////////////////////////////
/////////////Testing Cohap Related Vars////////////////////////////////////
///////////////////////////////////////////////////////////////////////////

	//Initialize Only	
	MyCohapTest : FB_COHAP;
	bInitializeCohapSystem: BOOL;
	bRes_CohapConnected: BOOL;

//	//Execute RunImpMethods Only	;
	bExecuteRunImpMethods: BOOL;
	bRes_RunImpMethods: BOOL;

//	//Set Current Device Instance
	bSetCurrentDevice_Cohap : BOOL;
	bRes_SetCurrentDevice : BOOL;
//	//Input Params
	strDeviceName : STRING;
	
	//RunCommand
	bRunCommandCohapSystem : BOOL;
	bRes_RunCommand : BOOL;
	
	//Input Params
	strMethodName : STRING;
	RunCom_InpuParams : T_CohapParameterList;
	RunCom_ExpOutParamList : ARRAY[0..9] OF ST_ReturnParamsInfo;
	
	//Output Params
	RunCom_OutputParams : T_CohapParameterList;
	
	//DummyTest Dictionary Prep for RunCommand Execution
	RC_DT_InpPar : T_CohapParameterList;
	RC_DT_ExpOutPL : ARRAY[0..9] OF ST_ReturnParamsInfo;
	
	CohapMethodStrings : TMethodNames_Cohap;
	CohapMethodControls : TMethod_Controls;
//	fbCohapHandler1: FB_COHAP;

///////////////////////////////

	// For readSerialNumber
	readSerialNumber_inpuparams : T_CohapParameterList;
	readSerialNumber_expoutparamlist : ARRAY[0..9] OF ST_ReturnParamsInfo;
	readSerialNumber_outputparams : T_CohapParameterList;
	
	// For ReadDeviceOutput
	ReadDeviceOutput_inpuparams : T_CohapParameterList;
	ReadDeviceOutput_expoutparamlist : ARRAY[0..9] OF ST_ReturnParamsInfo;
	ReadDeviceOutput_outputparams : T_CohapParameterList;

	
	// For PowerUp
	PowerUp_inpuparams : T_CohapParameterList;
	PowerUp_expoutparamlist : ARRAY[0..9] OF ST_ReturnParamsInfo;
	PowerUp_outputparams : T_CohapParameterList;
	
	// For PowerDown
	PowerDown_inpuparams : T_CohapParameterList;
	PowerDown_expoutparamlist : ARRAY[0..9] OF ST_ReturnParamsInfo;
	PowerDown_outputparams : T_CohapParameterList;
	
	// For TestDummy
	TestDummy_inpuparams : T_CohapParameterList;
	TestDummy_expoutparamlist : ARRAY[0..9] OF ST_ReturnParamsInfo;
	TestDummy_outputparams : T_CohapParameterList;
	
	// For TestDummy2
	TestDummy2_inpuparams : T_CohapParameterList;
	TestDummy2_expoutparamlist : ARRAY[0..9] OF ST_ReturnParamsInfo;
	TestDummy2_outputparams : T_CohapParameterList;
	
	// For init
	init_inpuparams : T_CohapParameterList;
	init_expoutparamlist : ARRAY[0..9] OF ST_ReturnParamsInfo;
	init_outputparams : T_CohapParameterList;
	
	// For getSICAndChannelCardVersions
	getSICAndChannelCardVersions_inpuparams : T_CohapParameterList;
	getSICAndChannelCardVersions_expoutparamlist : ARRAY[0..9] OF ST_ReturnParamsInfo;
	getSICAndChannelCardVersions_outputparams : T_CohapParameterList;
	
	// For getDLLVersions
	getDLLVersions_inpuparams : T_CohapParameterList;
	getDLLVersions_expoutparamlist : ARRAY[0..9] OF ST_ReturnParamsInfo;
	getDLLVersions_outputparams : T_CohapParameterList;
	
	// For initDUT
	initDUT_inpuparams : T_CohapParameterList;
	initDUT_expoutparamlist : ARRAY[0..9] OF ST_ReturnParamsInfo;
	initDUT_outputparams : T_CohapParameterList;
	
	//For Fast Channel Data
	readFastChannelData_inputparams : T_CohapParameterList;
	readFastChannelData_expoutparamlist : ARRAY[0..9] OF ST_ReturnParamsInfo;
	readFastChannelData_outputparams : T_CohapParameterList;

	// For T1 Step 1 Calibration
	t1Step1_inpuparams : T_CohapParameterList;
	t1Step1_expoutparamlist : ARRAY[0..9] OF ST_ReturnParamsInfo;
	t1Step1_outputparams : T_CohapParameterList;
	
//	// For T1 Step 2 Calibration
//	t1Step2_inpuparams : T_CohapParameterList;
//	t1Step2_expoutparamlist : ARRAY[0..9] OF ST_ReturnParamsInfo;
//	t1Step2_outputparams : T_CohapParameterList;
	
//	// For T1 Step 3 Calibration
//	t1Step3_inpuparams : T_CohapParameterList;
//	t1Step3_expoutparamlist : ARRAY[0..9] OF ST_ReturnParamsInfo;
//	t1Step3_outputparams : T_CohapParameterList;
	
	// For T2 Step 1 Calibration
	t2Step1_inpuparams : T_CohapParameterList;
	t2Step1_expoutparamlist : ARRAY[0..9] OF ST_ReturnParamsInfo;
	t2Step1_outputparams : T_CohapParameterList;
	
	// For T2 Step 2 Calibration
	t2Step2_inpuparams : T_CohapParameterList;
	t2Step2_expoutparamlist : ARRAY[0..9] OF ST_ReturnParamsInfo;
	t2Step2_outputparams : T_CohapParameterList;
	
	// For T2 Step 3 Calibration
	t2Step3_inpuparams : T_CohapParameterList;
	t2Step3_expoutparamlist : ARRAY[0..9] OF ST_ReturnParamsInfo;
	t2Step3_outputparams : T_CohapParameterList;
	
	// InitLot Device12133 class in Mech Device Lib Calibration
	InitLot_inputparams : T_CohapParameterList;
	InitLot_expoutparamlist : ARRAY[0..9] OF ST_ReturnParamsInfo;
	InitLot_outputparams : T_CohapParameterList;
	
//	//For Init Lot
//	InitLot_inputparams : T_CohapParameterList;
//	InitLot_expoutparamlist : ARRAY[0..9] OF ST_ReturnParamsInfo;
//	InitLot_outputparams : T_CohapParameterList;	
	// For T1 Step 1 Calibration
	t1Precal_inputparams : T_CohapParameterList;
	t1Precal_expoutparamlist : ARRAY[0..9] OF ST_ReturnParamsInfo;
	t1Precal_outputparams : T_CohapParameterList;
	// For T1 Step 2 Calibration
	t1Step2_inputparams : T_CohapParameterList;
	t1Step2_expoutparamlist : ARRAY[0..9] OF ST_ReturnParamsInfo;
	t1Step2_outputparams : T_CohapParameterList;
	// For T1 Step 3 Calibration
	t1Step3_inputparams : T_CohapParameterList;
	t1Step3_expoutparamlist : ARRAY[0..9] OF ST_ReturnParamsInfo;
	t1Step3_outputparams : T_CohapParameterList;
	
END_VAR
VAR // added by the converter: edge detectors and wires of the graphical bodies
    _w1, _w2, _w3, _w4, _w5, _w6, _w7, _w8, _w9, _w10, _w11, _w12, _w13, _w14, _w15, _w16, _w17, _w18, _w19, _w20, _w21, _w22, _w23, _w24, _w25, _w26, _w27, _w28, _w29, _w30, _w31, _w32, _w33, _w34, _w35, _w36, _w37, _w38, _w39, _w40 : BOOL;
END_VAR

bTestOutput := bTestInput;

A_Machine();
M_TestMESVars();
M_TestLaserMarker();
M_TestCohapLibrary();
//A_CohapLibraryTesting();
//A_InitCohapMethodParams();
//A_CohapLDTesting();

//A_Station1();
//A_Station2();
//A_Station3();
//A_Station4();
//bInterfaceTest := MyLaser1.fbApi.P_bDeviceInterfaceBusy;



//IF bPerformGetLotInfoFromLotBarcode THEN
//	_inst_bGetLotInfo_LotBarcode := fbDataHandler3.M_TransferData(in_strParamDBName_GetLotInfo);
//	IF _inst_bGetLotInfo_LotBarcode THEN
//		bPerformGetLotInfoFromLotBarcode := FALSE;
//	ELSIF fbDataHandler3.P_bError THEN 
//		bPerformGetLotInfoFromLotBarcode := FALSE;
//		fbDataHandler3.M_ClearError();
//	END_IF
//END_IF

//IF bPerformGetOpInfoFromOpBarcode THEN
//	_inst_bGetOpInfo_OpBarcode := fbDataHandler3.M_TransferData(in_strParamDBName_GetOpInfo);
//	IF _inst_bGetOpInfo_OpBarcode THEN
//		bPerformGetOpInfoFromOpBarcode := FALSE;
//	ELSIF fbDataHandler3.P_bError THEN 
//		bPerformGetOpInfoFromOpBarcode := FALSE;
//		fbDataHandler3.M_ClearError();
//	END_IF
//END_IF

//IF bPerformStartLot THEN
//	_inst_bStartLot := fbDataHandler3.M_TransferData(in_strParamDBName_StartLot);
//	IF _inst_bStartLot THEN
//		bPerformStartLot := FALSE;
//	ELSIF fbDataHandler3.P_bError THEN 
//		bPerformStartLot := FALSE;
//		fbDataHandler3.M_ClearError();
//	END_IF
//END_IF

//IF bPerformGetProdLotComponents THEN
//	_inst_bGetProdLotComponents := fbDataHandler3.M_TransferData(in_strParamDBName_GetProdLotComps);
//	IF _inst_bGetProdLotComponents THEN
//		bPerformGetProdLotComponents := FALSE;
//	ELSIF fbDataHandler3.P_bError THEN 
//		bPerformGetProdLotComponents := FALSE;
//		fbDataHandler3.M_ClearError();
//	END_IF
//END_IF


//IF bPerformComponentValidation1 THEN
//	_inst_bCompValidation1 := fbDataHandler3.M_TransferData(in_strParamDBName_Comp1Validation1);
//	IF _inst_bCompValidation1 THEN
//		bPerformComponentValidation1 := FALSE;
//	ELSIF fbDataHandler3.P_bError THEN 
//		bPerformComponentValidation1 := FALSE;
//		fbDataHandler3.M_ClearError();
//	END_IF
//END_IF

//IF bPerformComponentValidation2 THEN
//	_inst_bCompValidation2 := fbDataHandler3.M_TransferData(in_strParamDBName_Comp1Validation2);
//	IF _inst_bCompValidation2 THEN
//		bPerformComponentValidation2 := FALSE;
//	ELSIF fbDataHandler3.P_bError THEN 
//		bPerformComponentValidation2 := FALSE;
//		fbDataHandler3.M_ClearError();
//	END_IF
//END_IF

//IF bPerformComponentValidation3 THEN
//	_inst_bCompValidation3 := fbDataHandler3.M_TransferData(in_strParamDBName_Comp1Validation3);
//	IF _inst_bCompValidation3 THEN
//		bPerformComponentValidation3 := FALSE;
//	ELSIF fbDataHandler3.P_bError THEN 
//		bPerformComponentValidation3 := FALSE;
//		fbDataHandler3.M_ClearError();
//	END_IF
//END_IF

//IF bPerformGetMachineSettings THEN
//	_inst_bGetMachineSettings := fbDataHandler3.M_TransferData(in_strParamDBName_GetMachSetting);
//	IF _inst_bGetMachineSettings THEN
//		bPerformGetMachineSettings := FALSE;
//	ELSIF fbDataHandler3.P_bError THEN 
//		bPerformGetMachineSettings := FALSE;
//		fbDataHandler3.M_ClearError();
//	END_IF
//END_IF

//IF bPerformAddScrapCompByReason THEN
//	_inst_bAddScrapCompByReason := fbDataHandler3.M_TransferData(in_strParamDBName_AddScrapCompByReason);
//	IF _inst_bAddScrapCompByReason THEN
//		bPerformAddScrapCompByReason := FALSE;
//	ELSIF fbDataHandler3.P_bError THEN 
//		bPerformAddScrapCompByReason := FALSE;
//		fbDataHandler3.M_ClearError();
//	END_IF
//END_IF

//IF bPerformEndLotComp THEN
//	_inst_bEndLotComp := fbDataHandler3.M_TransferData(in_strParamDBName_EndLotComp);
//	IF _inst_bEndLotComp THEN
//		bPerformEndLotComp := FALSE;
//	ELSIF fbDataHandler3.P_bError THEN 
//		bPerformEndLotComp := FALSE;
//		fbDataHandler3.M_ClearError();
//	END_IF
//END_IF

//IF bPerformGetMachineDefects THEN
//	_inst_bGetMachineDefects := fbDataHandler3.M_TransferData(in_strParamDBName_GetMachDefects);
//	IF _inst_bGetMachineDefects THEN
//		bPerformGetMachineDefects := FALSE;
//	ELSIF fbDataHandler3.P_bError THEN 
//		bPerformGetMachineDefects := FALSE;
//		fbDataHandler3.M_ClearError();
//	END_IF
//END_IF

ACTION A_CohapLDTesting:
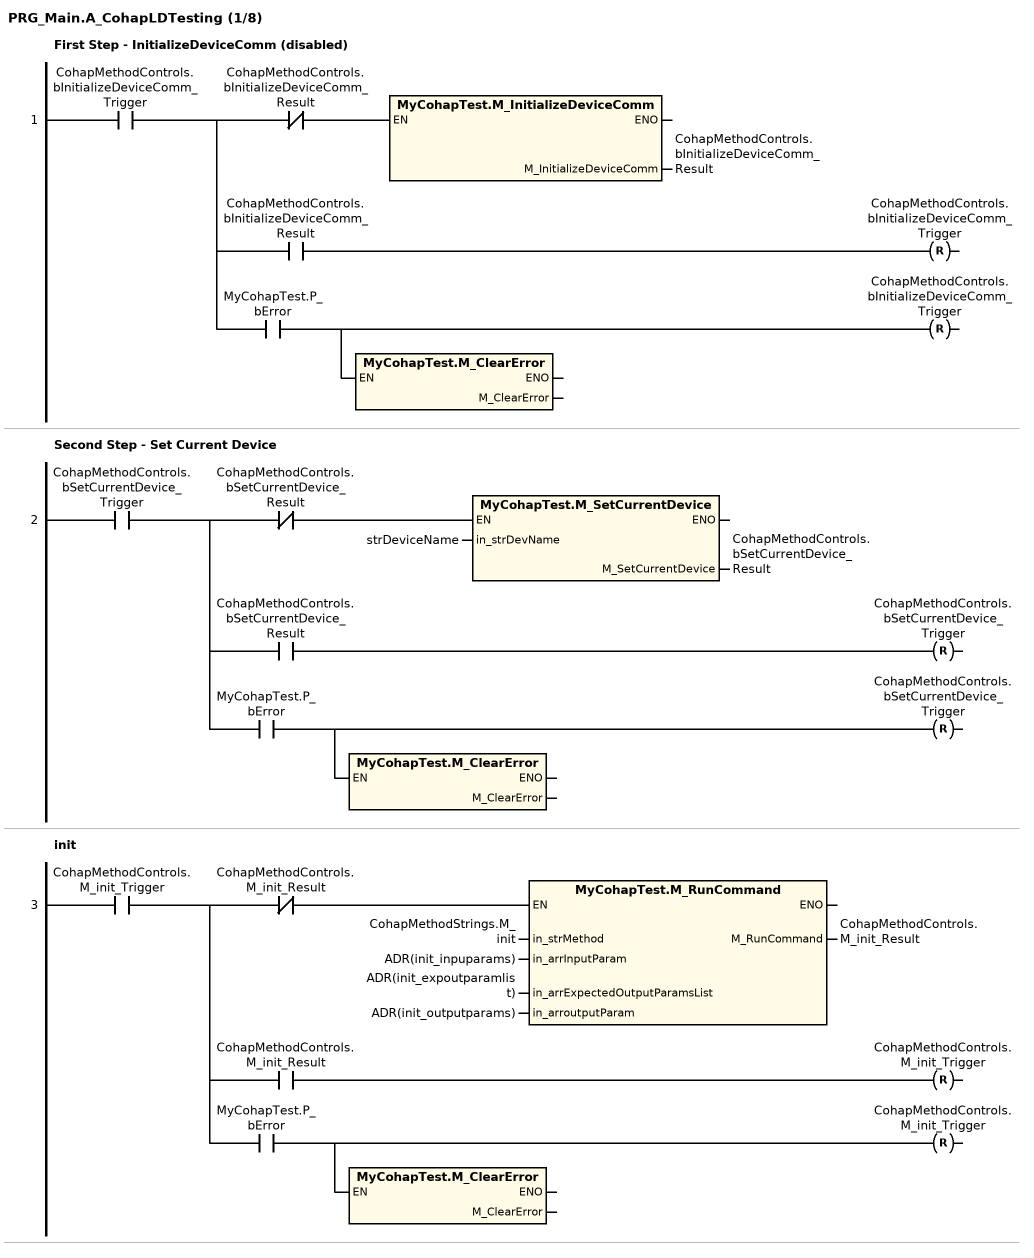
// NETWORK 1: First Step - InitializeDeviceComm (disabled)
// _w1 := CohapMethodControls.bInitializeDeviceComm_Trigger;
// IF _w1 AND NOT CohapMethodControls.bInitializeDeviceComm_Result THEN
//     CohapMethodControls.bInitializeDeviceComm_Result := MyCohapTest.M_InitializeDeviceComm();
// END_IF
// CohapMethodControls.bInitializeDeviceComm_Trigger R= _w1 AND CohapMethodControls.bInitializeDeviceComm_Result;
// _w2 := _w1 AND MyCohapTest.P_bError;
// CohapMethodControls.bInitializeDeviceComm_Trigger R= _w2;
// IF _w2 THEN MyCohapTest.M_ClearError(); END_IF

// NETWORK 2: Second Step - Set Current Device
_w3 := CohapMethodControls.bSetCurrentDevice_Trigger;
IF _w3 AND NOT CohapMethodControls.bSetCurrentDevice_Result THEN
    CohapMethodControls.bSetCurrentDevice_Result := MyCohapTest.M_SetCurrentDevice(in_strDevName := strDeviceName);
END_IF
CohapMethodControls.bSetCurrentDevice_Trigger R= _w3 AND CohapMethodControls.bSetCurrentDevice_Result;
_w4 := _w3 AND MyCohapTest.P_bError;
CohapMethodControls.bSetCurrentDevice_Trigger R= _w4;
IF _w4 THEN MyCohapTest.M_ClearError(); END_IF

// NETWORK 3: init
_w5 := CohapMethodControls.M_init_Trigger;
IF _w5 AND NOT CohapMethodControls.M_init_Result THEN
    CohapMethodControls.M_init_Result := MyCohapTest.M_RunCommand(in_strMethod := CohapMethodStrings.M_init, in_arrInputParam := ADR(init_inpuparams), in_arrExpectedOutputParamsList := ADR(init_expoutparamlist), in_arroutputParam := ADR(init_outputparams));
END_IF
CohapMethodControls.M_init_Trigger R= _w5 AND CohapMethodControls.M_init_Result;
_w6 := _w5 AND MyCohapTest.P_bError;
CohapMethodControls.M_init_Trigger R= _w6;
IF _w6 THEN MyCohapTest.M_ClearError(); END_IF

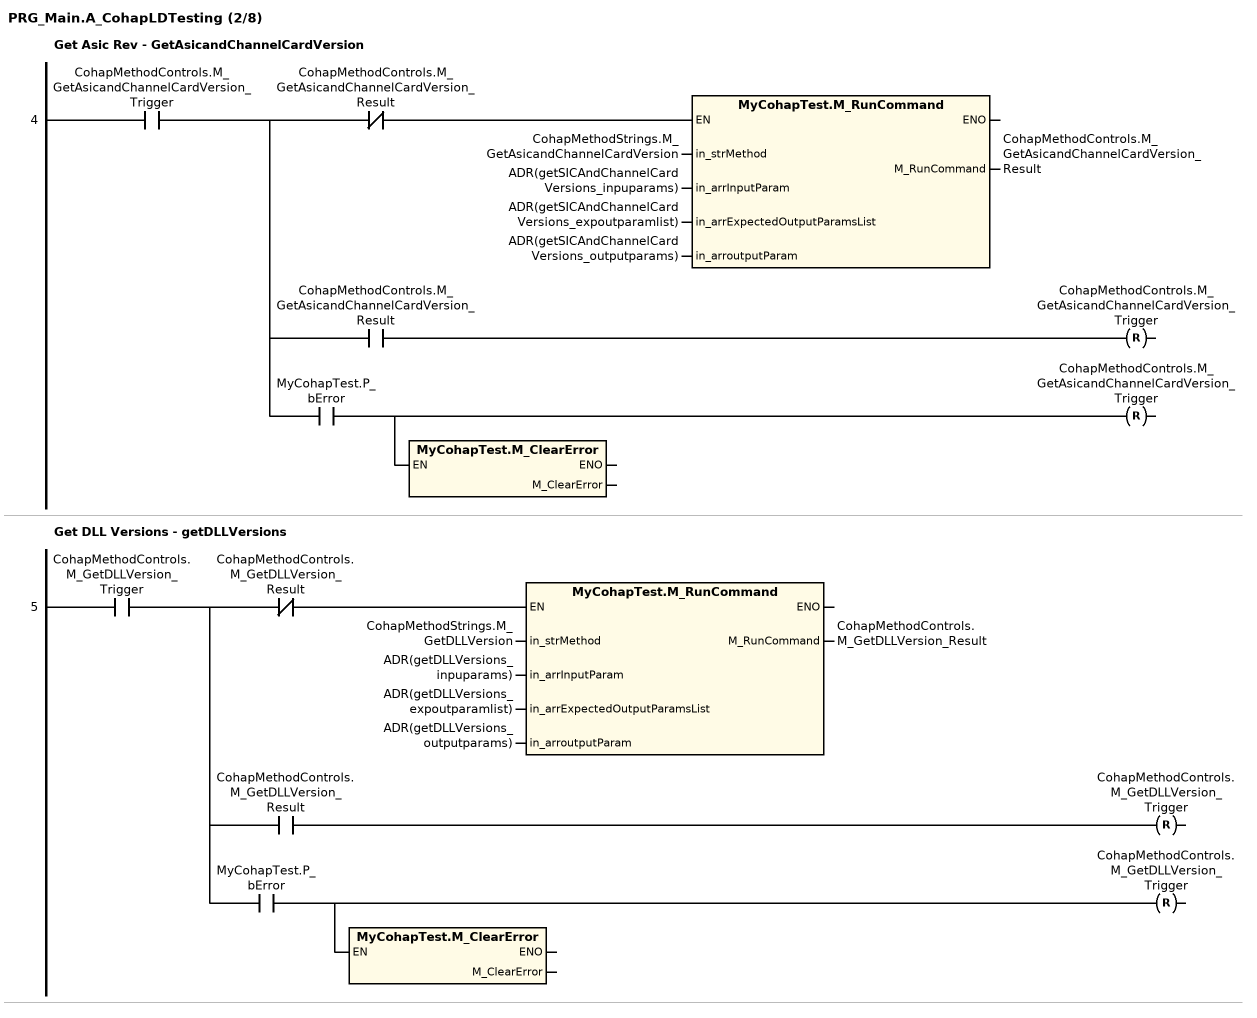
// NETWORK 4: Get Asic Rev - GetAsicandChannelCardVersion
_w7 := CohapMethodControls.M_GetAsicandChannelCardVersion_Trigger;
IF _w7 AND NOT CohapMethodControls.M_GetAsicandChannelCardVersion_Result THEN
    CohapMethodControls.M_GetAsicandChannelCardVersion_Result := MyCohapTest.M_RunCommand(in_strMethod := CohapMethodStrings.M_GetAsicandChannelCardVersion, in_arrInputParam := ADR(getSICAndChannelCardVersions_inpuparams), in_arrExpectedOutputParamsList := ADR(getSICAndChannelCardVersions_expoutparamlist), in_arroutputParam := ADR(getSICAndChannelCardVersions_outputparams));
END_IF
CohapMethodControls.M_GetAsicandChannelCardVersion_Trigger R= _w7 AND CohapMethodControls.M_GetAsicandChannelCardVersion_Result;
_w8 := _w7 AND MyCohapTest.P_bError;
CohapMethodControls.M_GetAsicandChannelCardVersion_Trigger R= _w8;
IF _w8 THEN MyCohapTest.M_ClearError(); END_IF

// NETWORK 5: Get DLL Versions - getDLLVersions
_w9 := CohapMethodControls.M_GetDLLVersion_Trigger;
IF _w9 AND NOT CohapMethodControls.M_GetDLLVersion_Result THEN
    CohapMethodControls.M_GetDLLVersion_Result := MyCohapTest.M_RunCommand(in_strMethod := CohapMethodStrings.M_GetDLLVersion, in_arrInputParam := ADR(getDLLVersions_inpuparams), in_arrExpectedOutputParamsList := ADR(getDLLVersions_expoutparamlist), in_arroutputParam := ADR(getDLLVersions_outputparams));
END_IF
CohapMethodControls.M_GetDLLVersion_Trigger R= _w9 AND CohapMethodControls.M_GetDLLVersion_Result;
_w10 := _w9 AND MyCohapTest.P_bError;
CohapMethodControls.M_GetDLLVersion_Trigger R= _w10;
IF _w10 THEN MyCohapTest.M_ClearError(); END_IF

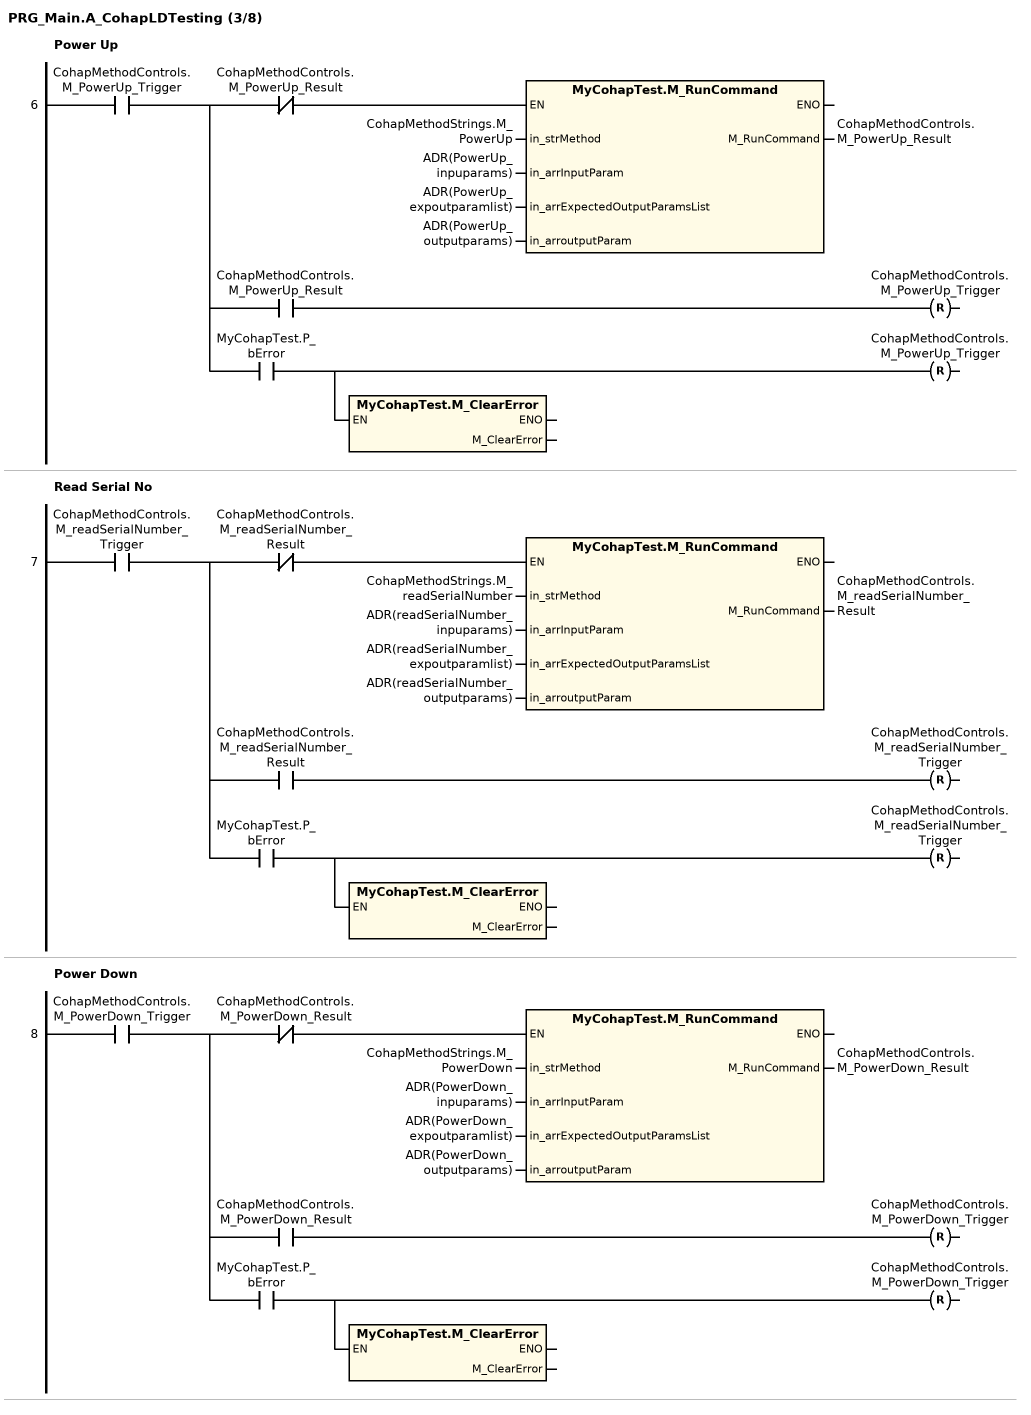
// NETWORK 6: Power Up
_w11 := CohapMethodControls.M_PowerUp_Trigger;
IF _w11 AND NOT CohapMethodControls.M_PowerUp_Result THEN
    CohapMethodControls.M_PowerUp_Result := MyCohapTest.M_RunCommand(in_strMethod := CohapMethodStrings.M_PowerUp, in_arrInputParam := ADR(PowerUp_inpuparams), in_arrExpectedOutputParamsList := ADR(PowerUp_expoutparamlist), in_arroutputParam := ADR(PowerUp_outputparams));
END_IF
CohapMethodControls.M_PowerUp_Trigger R= _w11 AND CohapMethodControls.M_PowerUp_Result;
_w12 := _w11 AND MyCohapTest.P_bError;
CohapMethodControls.M_PowerUp_Trigger R= _w12;
IF _w12 THEN MyCohapTest.M_ClearError(); END_IF

// NETWORK 7: Read Serial No
_w13 := CohapMethodControls.M_readSerialNumber_Trigger;
IF _w13 AND NOT CohapMethodControls.M_readSerialNumber_Result THEN
    CohapMethodControls.M_readSerialNumber_Result := MyCohapTest.M_RunCommand(in_strMethod := CohapMethodStrings.M_readSerialNumber, in_arrInputParam := ADR(readSerialNumber_inpuparams), in_arrExpectedOutputParamsList := ADR(readSerialNumber_expoutparamlist), in_arroutputParam := ADR(readSerialNumber_outputparams));
END_IF
CohapMethodControls.M_readSerialNumber_Trigger R= _w13 AND CohapMethodControls.M_readSerialNumber_Result;
_w14 := _w13 AND MyCohapTest.P_bError;
CohapMethodControls.M_readSerialNumber_Trigger R= _w14;
IF _w14 THEN MyCohapTest.M_ClearError(); END_IF

// NETWORK 8: Power Down
_w15 := CohapMethodControls.M_PowerDown_Trigger;
IF _w15 AND NOT CohapMethodControls.M_PowerDown_Result THEN
    CohapMethodControls.M_PowerDown_Result := MyCohapTest.M_RunCommand(in_strMethod := CohapMethodStrings.M_PowerDown, in_arrInputParam := ADR(PowerDown_inpuparams), in_arrExpectedOutputParamsList := ADR(PowerDown_expoutparamlist), in_arroutputParam := ADR(PowerDown_outputparams));
END_IF
CohapMethodControls.M_PowerDown_Trigger R= _w15 AND CohapMethodControls.M_PowerDown_Result;
_w16 := _w15 AND MyCohapTest.P_bError;
CohapMethodControls.M_PowerDown_Trigger R= _w16;
IF _w16 THEN MyCohapTest.M_ClearError(); END_IF

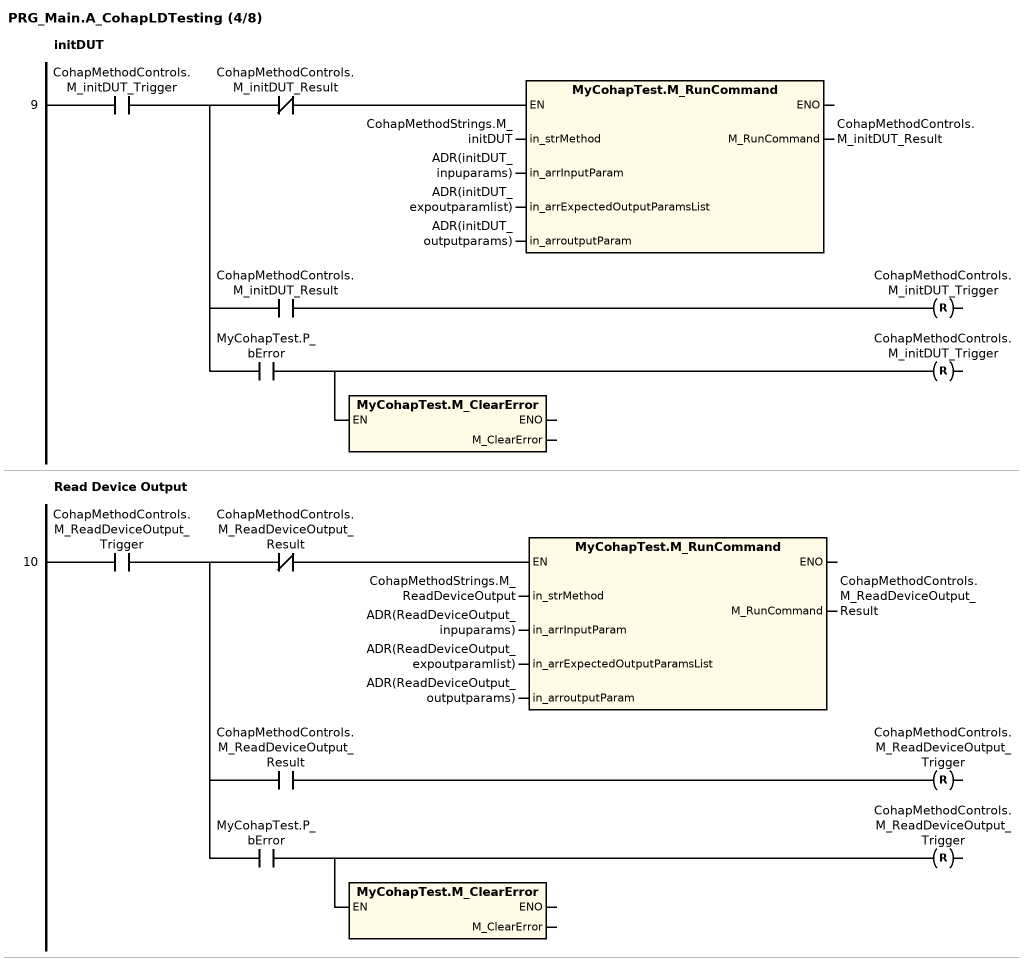
// NETWORK 9: initDUT
_w17 := CohapMethodControls.M_initDUT_Trigger;
IF _w17 AND NOT CohapMethodControls.M_initDUT_Result THEN
    CohapMethodControls.M_initDUT_Result := MyCohapTest.M_RunCommand(in_strMethod := CohapMethodStrings.M_initDUT, in_arrInputParam := ADR(initDUT_inpuparams), in_arrExpectedOutputParamsList := ADR(initDUT_expoutparamlist), in_arroutputParam := ADR(initDUT_outputparams));
END_IF
CohapMethodControls.M_initDUT_Trigger R= _w17 AND CohapMethodControls.M_initDUT_Result;
_w18 := _w17 AND MyCohapTest.P_bError;
CohapMethodControls.M_initDUT_Trigger R= _w18;
IF _w18 THEN MyCohapTest.M_ClearError(); END_IF

// NETWORK 10: Read Device Output
_w19 := CohapMethodControls.M_ReadDeviceOutput_Trigger;
IF _w19 AND NOT CohapMethodControls.M_ReadDeviceOutput_Result THEN
    CohapMethodControls.M_ReadDeviceOutput_Result := MyCohapTest.M_RunCommand(in_strMethod := CohapMethodStrings.M_ReadDeviceOutput, in_arrInputParam := ADR(ReadDeviceOutput_inpuparams), in_arrExpectedOutputParamsList := ADR(ReadDeviceOutput_expoutparamlist), in_arroutputParam := ADR(ReadDeviceOutput_outputparams));
END_IF
CohapMethodControls.M_ReadDeviceOutput_Trigger R= _w19 AND CohapMethodControls.M_ReadDeviceOutput_Result;
_w20 := _w19 AND MyCohapTest.P_bError;
CohapMethodControls.M_ReadDeviceOutput_Trigger R= _w20;
IF _w20 THEN MyCohapTest.M_ClearError(); END_IF

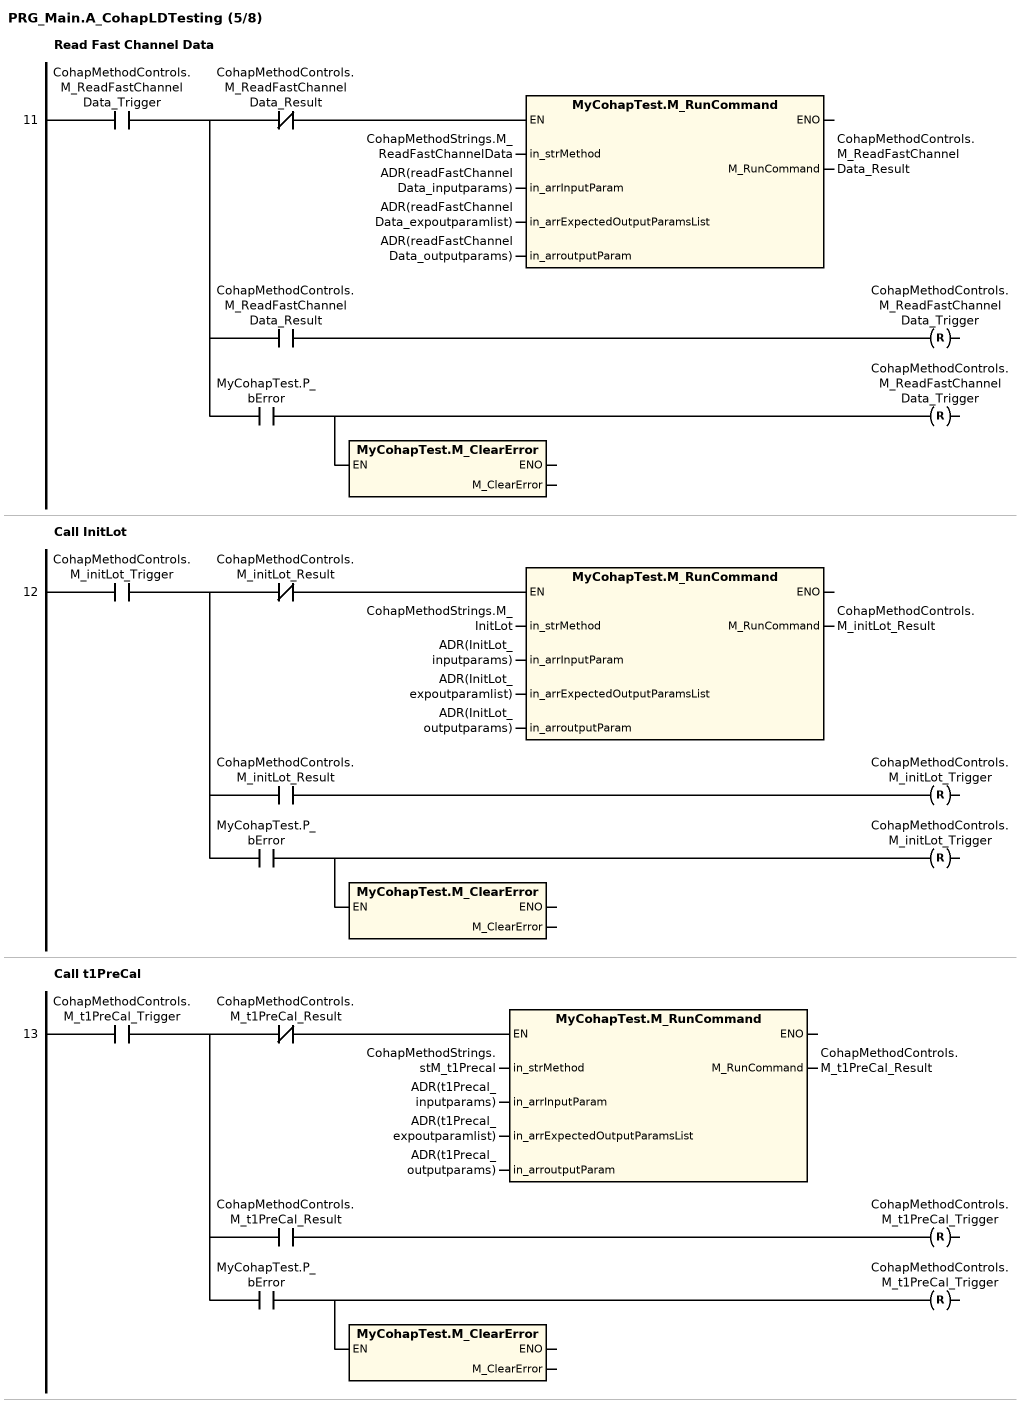
// NETWORK 11: Read Fast Channel Data
_w21 := CohapMethodControls.M_ReadFastChannelData_Trigger;
IF _w21 AND NOT CohapMethodControls.M_ReadFastChannelData_Result THEN
    CohapMethodControls.M_ReadFastChannelData_Result := MyCohapTest.M_RunCommand(in_strMethod := CohapMethodStrings.M_ReadFastChannelData, in_arrInputParam := ADR(readFastChannelData_inputparams), in_arrExpectedOutputParamsList := ADR(readFastChannelData_expoutparamlist), in_arroutputParam := ADR(readFastChannelData_outputparams));
END_IF
CohapMethodControls.M_ReadFastChannelData_Trigger R= _w21 AND CohapMethodControls.M_ReadFastChannelData_Result;
_w22 := _w21 AND MyCohapTest.P_bError;
CohapMethodControls.M_ReadFastChannelData_Trigger R= _w22;
IF _w22 THEN MyCohapTest.M_ClearError(); END_IF

// NETWORK 12: Call InitLot
_w23 := CohapMethodControls.M_initLot_Trigger;
IF _w23 AND NOT CohapMethodControls.M_initLot_Result THEN
    CohapMethodControls.M_initLot_Result := MyCohapTest.M_RunCommand(in_strMethod := CohapMethodStrings.M_InitLot, in_arrInputParam := ADR(InitLot_inputparams), in_arrExpectedOutputParamsList := ADR(InitLot_expoutparamlist), in_arroutputParam := ADR(InitLot_outputparams));
END_IF
CohapMethodControls.M_initLot_Trigger R= _w23 AND CohapMethodControls.M_initLot_Result;
_w24 := _w23 AND MyCohapTest.P_bError;
CohapMethodControls.M_initLot_Trigger R= _w24;
IF _w24 THEN MyCohapTest.M_ClearError(); END_IF

// NETWORK 13: Call t1PreCal
_w25 := CohapMethodControls.M_t1PreCal_Trigger;
IF _w25 AND NOT CohapMethodControls.M_t1PreCal_Result THEN
    CohapMethodControls.M_t1PreCal_Result := MyCohapTest.M_RunCommand(in_strMethod := CohapMethodStrings.stM_t1Precal, in_arrInputParam := ADR(t1Precal_inputparams), in_arrExpectedOutputParamsList := ADR(t1Precal_expoutparamlist), in_arroutputParam := ADR(t1Precal_outputparams));
END_IF
CohapMethodControls.M_t1PreCal_Trigger R= _w25 AND CohapMethodControls.M_t1PreCal_Result;
_w26 := _w25 AND MyCohapTest.P_bError;
CohapMethodControls.M_t1PreCal_Trigger R= _w26;
IF _w26 THEN MyCohapTest.M_ClearError(); END_IF

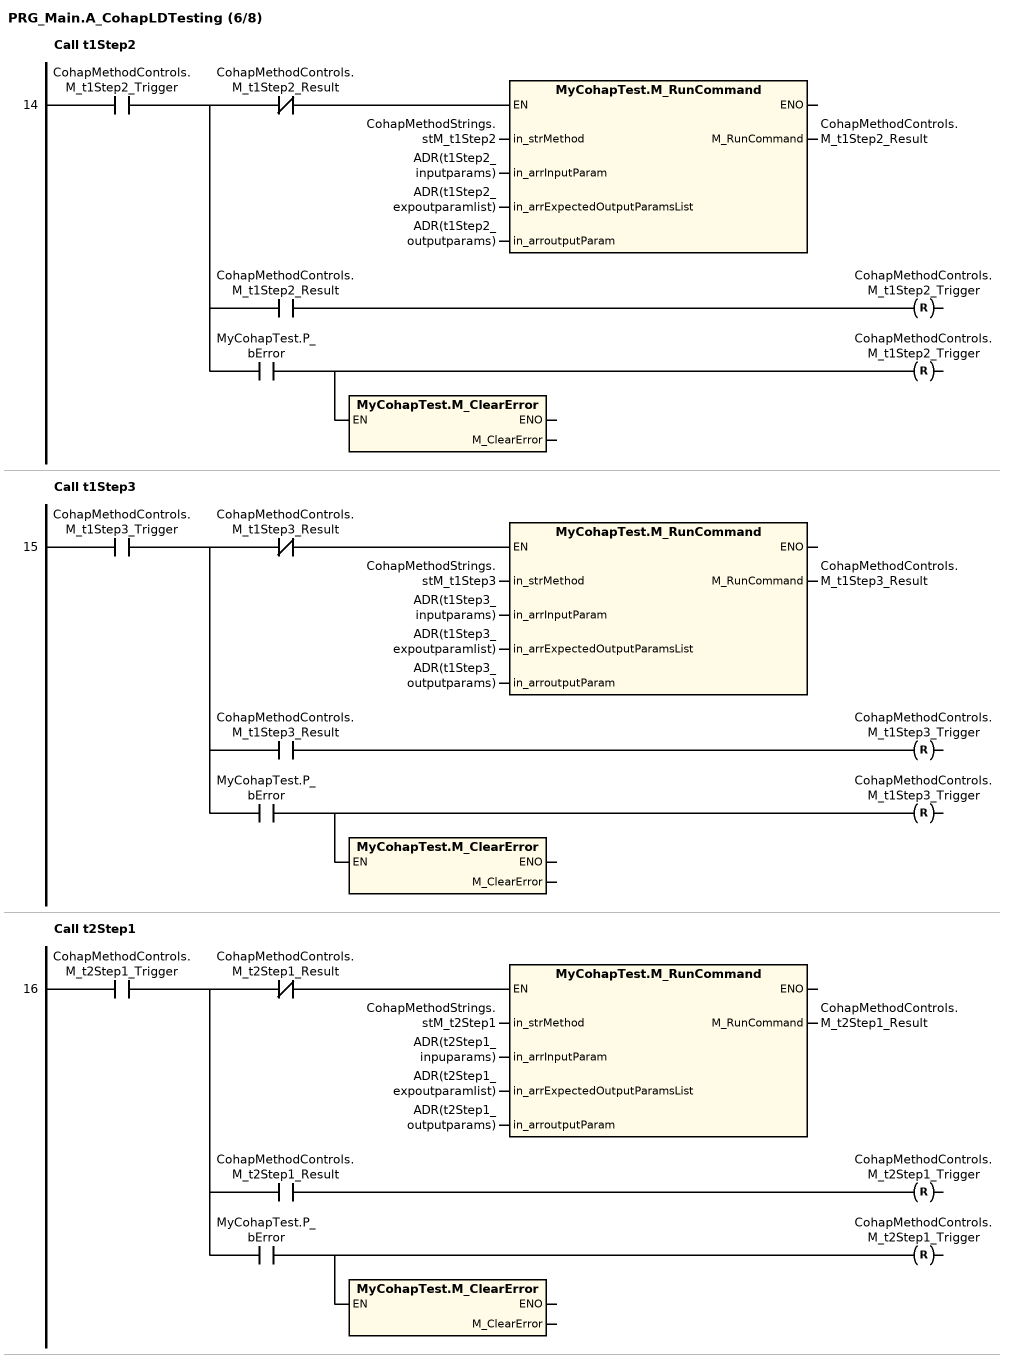
// NETWORK 14: Call t1Step2
_w27 := CohapMethodControls.M_t1Step2_Trigger;
IF _w27 AND NOT CohapMethodControls.M_t1Step2_Result THEN
    CohapMethodControls.M_t1Step2_Result := MyCohapTest.M_RunCommand(in_strMethod := CohapMethodStrings.stM_t1Step2, in_arrInputParam := ADR(t1Step2_inputparams), in_arrExpectedOutputParamsList := ADR(t1Step2_expoutparamlist), in_arroutputParam := ADR(t1Step2_outputparams));
END_IF
CohapMethodControls.M_t1Step2_Trigger R= _w27 AND CohapMethodControls.M_t1Step2_Result;
_w28 := _w27 AND MyCohapTest.P_bError;
CohapMethodControls.M_t1Step2_Trigger R= _w28;
IF _w28 THEN MyCohapTest.M_ClearError(); END_IF

// NETWORK 15: Call t1Step3
_w29 := CohapMethodControls.M_t1Step3_Trigger;
IF _w29 AND NOT CohapMethodControls.M_t1Step3_Result THEN
    CohapMethodControls.M_t1Step3_Result := MyCohapTest.M_RunCommand(in_strMethod := CohapMethodStrings.stM_t1Step3, in_arrInputParam := ADR(t1Step3_inputparams), in_arrExpectedOutputParamsList := ADR(t1Step3_expoutparamlist), in_arroutputParam := ADR(t1Step3_outputparams));
END_IF
CohapMethodControls.M_t1Step3_Trigger R= _w29 AND CohapMethodControls.M_t1Step3_Result;
_w30 := _w29 AND MyCohapTest.P_bError;
CohapMethodControls.M_t1Step3_Trigger R= _w30;
IF _w30 THEN MyCohapTest.M_ClearError(); END_IF

// NETWORK 16: Call t2Step1
_w31 := CohapMethodControls.M_t2Step1_Trigger;
IF _w31 AND NOT CohapMethodControls.M_t2Step1_Result THEN
    CohapMethodControls.M_t2Step1_Result := MyCohapTest.M_RunCommand(in_strMethod := CohapMethodStrings.stM_t2Step1, in_arrInputParam := ADR(t2Step1_inpuparams), in_arrExpectedOutputParamsList := ADR(t2Step1_expoutparamlist), in_arroutputParam := ADR(t2Step1_outputparams));
END_IF
CohapMethodControls.M_t2Step1_Trigger R= _w31 AND CohapMethodControls.M_t2Step1_Result;
_w32 := _w31 AND MyCohapTest.P_bError;
CohapMethodControls.M_t2Step1_Trigger R= _w32;
IF _w32 THEN MyCohapTest.M_ClearError(); END_IF

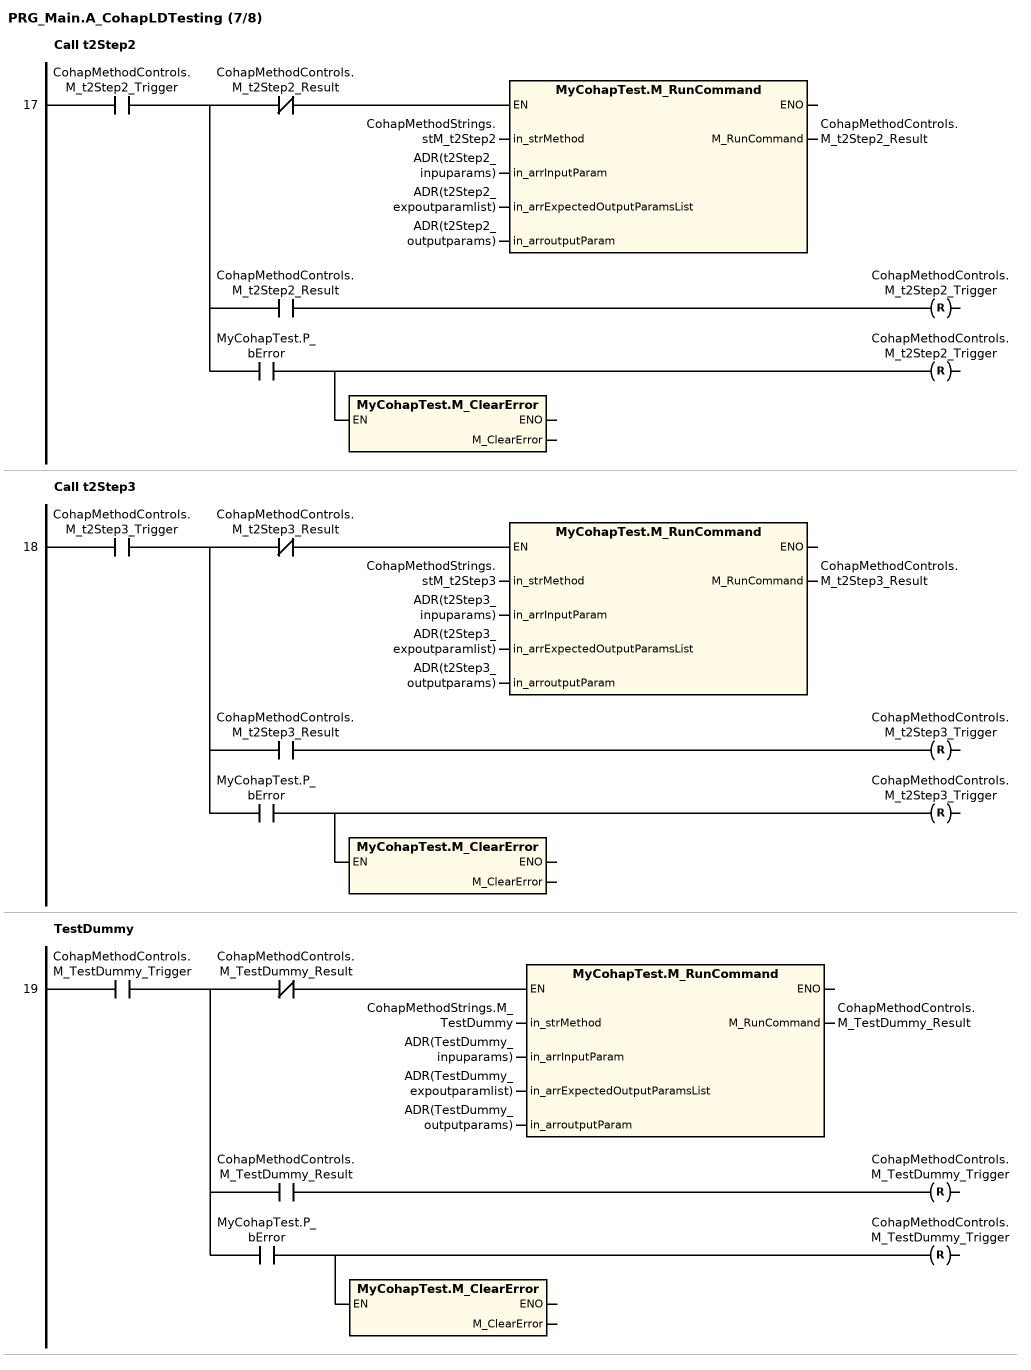
// NETWORK 17: Call t2Step2
_w33 := CohapMethodControls.M_t2Step2_Trigger;
IF _w33 AND NOT CohapMethodControls.M_t2Step2_Result THEN
    CohapMethodControls.M_t2Step2_Result := MyCohapTest.M_RunCommand(in_strMethod := CohapMethodStrings.stM_t2Step2, in_arrInputParam := ADR(t2Step2_inpuparams), in_arrExpectedOutputParamsList := ADR(t2Step2_expoutparamlist), in_arroutputParam := ADR(t2Step2_outputparams));
END_IF
CohapMethodControls.M_t2Step2_Trigger R= _w33 AND CohapMethodControls.M_t2Step2_Result;
_w34 := _w33 AND MyCohapTest.P_bError;
CohapMethodControls.M_t2Step2_Trigger R= _w34;
IF _w34 THEN MyCohapTest.M_ClearError(); END_IF

// NETWORK 18: Call t2Step3
_w35 := CohapMethodControls.M_t2Step3_Trigger;
IF _w35 AND NOT CohapMethodControls.M_t2Step3_Result THEN
    CohapMethodControls.M_t2Step3_Result := MyCohapTest.M_RunCommand(in_strMethod := CohapMethodStrings.stM_t2Step3, in_arrInputParam := ADR(t2Step3_inpuparams), in_arrExpectedOutputParamsList := ADR(t2Step3_expoutparamlist), in_arroutputParam := ADR(t2Step3_outputparams));
END_IF
CohapMethodControls.M_t2Step3_Trigger R= _w35 AND CohapMethodControls.M_t2Step3_Result;
_w36 := _w35 AND MyCohapTest.P_bError;
CohapMethodControls.M_t2Step3_Trigger R= _w36;
IF _w36 THEN MyCohapTest.M_ClearError(); END_IF

// NETWORK 19: TestDummy
_w37 := CohapMethodControls.M_TestDummy_Trigger;
IF _w37 AND NOT CohapMethodControls.M_TestDummy_Result THEN
    CohapMethodControls.M_TestDummy_Result := MyCohapTest.M_RunCommand(in_strMethod := CohapMethodStrings.M_TestDummy, in_arrInputParam := ADR(TestDummy_inpuparams), in_arrExpectedOutputParamsList := ADR(TestDummy_expoutparamlist), in_arroutputParam := ADR(TestDummy_outputparams));
END_IF
CohapMethodControls.M_TestDummy_Trigger R= _w37 AND CohapMethodControls.M_TestDummy_Result;
_w38 := _w37 AND MyCohapTest.P_bError;
CohapMethodControls.M_TestDummy_Trigger R= _w38;
IF _w38 THEN MyCohapTest.M_ClearError(); END_IF

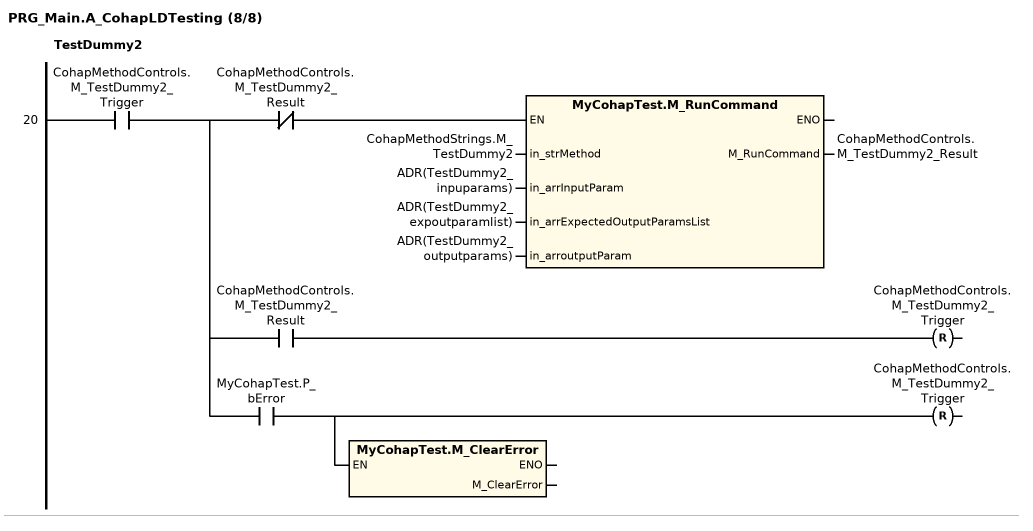
// NETWORK 20: TestDummy2
_w39 := CohapMethodControls.M_TestDummy2_Trigger;
IF _w39 AND NOT CohapMethodControls.M_TestDummy2_Result THEN
    CohapMethodControls.M_TestDummy2_Result := MyCohapTest.M_RunCommand(in_strMethod := CohapMethodStrings.M_TestDummy2, in_arrInputParam := ADR(TestDummy2_inpuparams), in_arrExpectedOutputParamsList := ADR(TestDummy2_expoutparamlist), in_arroutputParam := ADR(TestDummy2_outputparams));
END_IF
CohapMethodControls.M_TestDummy2_Trigger R= _w39 AND CohapMethodControls.M_TestDummy2_Result;
_w40 := _w39 AND MyCohapTest.P_bError;
CohapMethodControls.M_TestDummy2_Trigger R= _w40;
IF _w40 THEN MyCohapTest.M_ClearError(); END_IF
END_ACTION

ACTION A_CohapLibraryTesting:
//IF bInitializeCohapSystem THEN
//	bRes_CohapConnected := MyCohapTest.M_init(1);
//	IF bRes_CohapConnected THEN
//	//Add some timer based logic to do error handling.
//		bInitializeCohapSystem := FALSE;
//	ELSIF MyCohapTest.P_bError THEN
//		bInitializeCohapSystem := FALSE;
//		MyCohapTest.M_ClearError();
//	END_IF
//END_IF

//IF bExecuteRunImpMethods THEN
//	bRes_RunImpMethods := MyCohapTest.M_RunImpMethods();
//	IF bRes_RunImpMethods THEN
//	//Add some timer based logic to do error handling.
//		bExecuteRunImpMethods := FALSE;
//	ELSIF MyCohapTest.P_bError THEN
//		bExecuteRunImpMethods := FALSE;
//		MyCohapTest.M_ClearError();
//	END_IF
//END_IF


//IF bSetCurrentDevice_Cohap THEN
//	bRes_SetCurrentDevice := MyCohapTest.M_SetCurrentDevice(strDeviceName);
//	IF bRes_SetCurrentDevice THEN
//	//Add some timer based logic to do error handling.
//		bSetCurrentDevice_Cohap := FALSE;
//	ELSIF MyCohapTest.P_bError THEN
//		bSetCurrentDevice_Cohap := FALSE;
//		MyCohapTest.M_ClearError();
//	END_IF
//END_IF


//RC_DT_InpPar[1].strKey := 'channel';
//RC_DT_InpPar[1].strValue := '123';

////RC_DT_InpPar[1].strKey := '';
////RC_DT_InpPar[1].strValue := '';

//RC_DT_ExpOutPL[1].VarName := 'serialno';
//RC_DT_ExpOutPL[1].DataType := E_DataType.DT_STRING;

////RC_DT_ExpOutPL[1].VarName := '';
////RC_DT_ExpOutPL[1].DataType := E_DataType.DT_BOOL;


//IF bRunCommandCohapSystem THEN
//	bRes_RunCommand := MyCohapTest.M_RunCommand(strMethodName, RunCom_InpuParams, RunCom_ExpOutParamList, aoutputParam => RunCom_OutputParams );
//	IF bRes_RunCommand THEN
//	//Add some timer based logic to do error handling.
//		bRunCommandCohapSystem := FALSE;
//	ELSIF MyCohapTest.P_bError THEN
//		bRunCommandCohapSystem := FALSE;
//		MyCohapTest.M_ClearError();
//	END_IF
//END_IF
END_ACTION

ACTION A_InitCohapMethodParams:
//M_TestCohapLibrary.strDeviceName := 'Device12133';

//M_TestCohapLibrary.readSerialNumber_inpuparams[0].strKey := 'channel';
//M_TestCohapLibrary.readSerialNumber_inpuparams[0].strValue := '1';
//M_TestCohapLibrary.readSerialNumber_inpuparams[1].strKey := '';
//M_TestCohapLibrary.readSerialNumber_inpuparams[1].strValue := '';
//M_TestCohapLibrary.readSerialNumber_inpuparams[2].strKey := '';
//M_TestCohapLibrary.readSerialNumber_inpuparams[2].strValue := '';

//M_TestCohapLibrary.readSerialNumber_expoutparamlist[0].enumDataType := E_DataType.DT_ULINT;
//M_TestCohapLibrary.readSerialNumber_expoutparamlist[0].strVarName := 'serialnumber';
//M_TestCohapLibrary.readSerialNumber_expoutparamlist[1].enumDataType := E_DataType.DT_STRING;
//M_TestCohapLibrary.readSerialNumber_expoutparamlist[1].strVarName := 'stringserialno';
//M_TestCohapLibrary.readSerialNumber_expoutparamlist[2].enumDataType := E_DataType.DT_STRING;
//M_TestCohapLibrary.readSerialNumber_expoutparamlist[2].strVarName := '';


//M_TestCohapLibrary.ReadDeviceOutput_inpuparams[0].strKey := 'channel';
//M_TestCohapLibrary.ReadDeviceOutput_inpuparams[0].strValue := '1';
//M_TestCohapLibrary.ReadDeviceOutput_inpuparams[1].strKey := '';
//M_TestCohapLibrary.ReadDeviceOutput_inpuparams[1].strValue := '';
//M_TestCohapLibrary.ReadDeviceOutput_inpuparams[2].strKey := '';
//M_TestCohapLibrary.ReadDeviceOutput_inpuparams[2].strValue := '';

//M_TestCohapLibrary.ReadDeviceOutput_expoutparamlist[0].enumDataType := E_DataType.DT_INT;
//M_TestCohapLibrary.ReadDeviceOutput_expoutparamlist[0].strVarName := 'P1data';
//M_TestCohapLibrary.ReadDeviceOutput_expoutparamlist[1].enumDataType := E_DataType.DT_INT;
//M_TestCohapLibrary.ReadDeviceOutput_expoutparamlist[1].strVarName := 'P1out';
//M_TestCohapLibrary.ReadDeviceOutput_expoutparamlist[2].enumDataType := E_DataType.DT_INT;
//M_TestCohapLibrary.ReadDeviceOutput_expoutparamlist[2].strVarName := 'P2data';
//M_TestCohapLibrary.ReadDeviceOutput_expoutparamlist[3].enumDataType := E_DataType.DT_INT;
//M_TestCohapLibrary.ReadDeviceOutput_expoutparamlist[3].strVarName := 'P2out';
//M_TestCohapLibrary.ReadDeviceOutput_expoutparamlist[4].enumDataType := E_DataType.DT_INT;
//M_TestCohapLibrary.ReadDeviceOutput_expoutparamlist[4].strVarName := 'T1data';
//M_TestCohapLibrary.ReadDeviceOutput_expoutparamlist[5].enumDataType := E_DataType.DT_INT;
//M_TestCohapLibrary.ReadDeviceOutput_expoutparamlist[5].strVarName := 'T1out';
//M_TestCohapLibrary.ReadDeviceOutput_expoutparamlist[6].enumDataType := E_DataType.DT_INT;
//M_TestCohapLibrary.ReadDeviceOutput_expoutparamlist[6].strVarName := 'T2data';
//M_TestCohapLibrary.ReadDeviceOutput_expoutparamlist[7].enumDataType := E_DataType.DT_INT;
//M_TestCohapLibrary.ReadDeviceOutput_expoutparamlist[7].strVarName := 'T2out';

//M_TestCohapLibrary.PowerUp_inpuparams[0].strKey := 'channel';
//M_TestCohapLibrary.PowerUp_inpuparams[0].strValue := '1';
//M_TestCohapLibrary.PowerUp_inpuparams[1].strKey := 'supplyVoltage';
//M_TestCohapLibrary.PowerUp_inpuparams[1].strValue := '5.0';
//M_TestCohapLibrary.PowerUp_inpuparams[2].strKey := '';
//M_TestCohapLibrary.PowerUp_inpuparams[2].strValue := '';

//M_TestCohapLibrary.PowerUp_expoutparamlist[0].enumDataType := E_DataType.DT_DOUBLE;
//M_TestCohapLibrary.PowerUp_expoutparamlist[0].strVarName := 'Vsupply';
//M_TestCohapLibrary.PowerUp_expoutparamlist[1].enumDataType := E_DataType.DT_DOUBLE;
//M_TestCohapLibrary.PowerUp_expoutparamlist[1].strVarName := 'current';
//M_TestCohapLibrary.PowerUp_expoutparamlist[2].enumDataType := E_DataType.DT_STRING;
//M_TestCohapLibrary.PowerUp_expoutparamlist[2].strVarName := '';
//M_TestCohapLibrary.
//M_TestCohapLibrary.PowerDown_inpuparams[0].strKey := 'channel';
//M_TestCohapLibrary.PowerDown_inpuparams[0].strValue := '1';
//M_TestCohapLibrary.PowerDown_inpuparams[1].strKey := '';
//M_TestCohapLibrary.PowerDown_inpuparams[1].strValue := '';
//M_TestCohapLibrary.PowerDown_inpuparams[2].strKey := '';
//M_TestCohapLibrary.PowerDown_inpuparams[2].strValue := '';

//M_TestCohapLibrary.PowerDown_expoutparamlist[0].enumDataType := E_DataType.DT_STRING;
//M_TestCohapLibrary.PowerDown_expoutparamlist[0].strVarName := '';
//M_TestCohapLibrary.PowerDown_expoutparamlist[1].enumDataType := E_DataType.DT_STRING;
//M_TestCohapLibrary.PowerDown_expoutparamlist[1].strVarName := '';
//M_TestCohapLibrary.PowerDown_expoutparamlist[2].enumDataType := E_DataType.DT_STRING;
//M_TestCohapLibrary.PowerDown_expoutparamlist[2].strVarName := '';

//M_TestCohapLibrary.TestDummy_inpuparams[0].strKey := 'channel';
//M_TestCohapLibrary.TestDummy_inpuparams[0].strValue := '1';
//M_TestCohapLibrary.TestDummy_inpuparams[1].strKey := 'bInput';
//M_TestCohapLibrary.TestDummy_inpuparams[1].strValue := 'FALSE';
//M_TestCohapLibrary.TestDummy_inpuparams[2].strKey := '';
//M_TestCohapLibrary.TestDummy_inpuparams[2].strValue := '';

//M_TestCohapLibrary.TestDummy_expoutparamlist[0].enumDataType := E_DataType.DT_STRING;
//M_TestCohapLibrary.TestDummy_expoutparamlist[0].strVarName := 'serialno';
//M_TestCohapLibrary.TestDummy_expoutparamlist[1].enumDataType := E_DataType.DT_DOUBLE;
//M_TestCohapLibrary.TestDummy_expoutparamlist[1].strVarName := 'Voltage';
//M_TestCohapLibrary.TestDummy_expoutparamlist[2].enumDataType := E_DataType.DT_BOOL;
//M_TestCohapLibrary.TestDummy_expoutparamlist[2].strVarName := 'MethodResponse';
//M_TestCohapLibrary.TestDummy_expoutparamlist[3].enumDataType := E_DataType.DT_UINT;
//M_TestCohapLibrary.TestDummy_expoutparamlist[3].strVarName := 'current';
//M_TestCohapLibrary.TestDummy_expoutparamlist[4].enumDataType := E_DataType.DT_STRING;
//M_TestCohapLibrary.TestDummy_expoutparamlist[4].strVarName := 'P1status';
//M_TestCohapLibrary.TestDummy_expoutparamlist[5].enumDataType := E_DataType.DT_STRING;
//M_TestCohapLibrary.TestDummy_expoutparamlist[5].strVarName := 'P2status';

//M_TestCohapLibrary.TestDummy2_inpuparams[0].strKey := 'channel';
//M_TestCohapLibrary.TestDummy2_inpuparams[0].strValue := '1';
//M_TestCohapLibrary.TestDummy2_inpuparams[1].strKey := 'Input2';
//M_TestCohapLibrary.TestDummy2_inpuparams[1].strValue := 'dummyimput2';
//M_TestCohapLibrary.TestDummy2_inpuparams[2].strKey := '';
//M_TestCohapLibrary.TestDummy2_inpuparams[2].strValue := '';

//M_TestCohapLibrary.TestDummy2_expoutparamlist[0].enumDataType := E_DataType.DT_INT;
//M_TestCohapLibrary.TestDummy2_expoutparamlist[0].strVarName := 'output1';
//M_TestCohapLibrary.TestDummy2_expoutparamlist[1].enumDataType := E_DataType.DT_STRING;
//M_TestCohapLibrary.TestDummy2_expoutparamlist[1].strVarName := 'output2';
//M_TestCohapLibrary.TestDummy2_expoutparamlist[2].enumDataType := E_DataType.DT_ULINT;
//M_TestCohapLibrary.TestDummy2_expoutparamlist[2].strVarName := 'fastchannel1';
//M_TestCohapLibrary.TestDummy2_expoutparamlist[3].enumDataType := E_DataType.DT_ULINT;
//M_TestCohapLibrary.TestDummy2_expoutparamlist[3].strVarName := 'fastchannel2';
//M_TestCohapLibrary.TestDummy2_expoutparamlist[4].enumDataType := E_DataType.DT_STRING;
//M_TestCohapLibrary.TestDummy2_expoutparamlist[4].strVarName := 'fastchannel3';
//M_TestCohapLibrary.TestDummy2_expoutparamlist[5].enumDataType := E_DataType.DT_INT;
//M_TestCohapLibrary.TestDummy2_expoutparamlist[5].strVarName := 'fastchannel4';
//M_TestCohapLibrary.TestDummy2_expoutparamlist[6].enumDataType := E_DataType.DT_ULINT;
//M_TestCohapLibrary.TestDummy2_expoutparamlist[6].strVarName := 'fastchannel5';
//M_TestCohapLibrary.TestDummy2_expoutparamlist[7].enumDataType := E_DataType.DT_ULINT;
//M_TestCohapLibrary.TestDummy2_expoutparamlist[7].strVarName := 'fastchannel6';
//M_TestCohapLibrary.TestDummy2_expoutparamlist[8].enumDataType := E_DataType.DT_STRING;
//M_TestCohapLibrary.TestDummy2_expoutparamlist[8].strVarName := 'fastchannel7';
//M_TestCohapLibrary.TestDummy2_expoutparamlist[9].enumDataType := E_DataType.DT_INT;
//M_TestCohapLibrary.TestDummy2_expoutparamlist[9].strVarName := 'fastchannel8';

////TestDummy2_outputparams[0].strKey := '';
////TestDummy2_outputparams[0].strValue := '';
////TestDummy2_outputparams[1].strKey := '';
////TestDummy2_outputparams[1].strValue := '';
////TestDummy2_outputparams[2].strKey := '';
////TestDummy2_outputparams[2].strValue := '';
////TestDummy2_outputparams[3].strKey := '';
////TestDummy2_outputparams[3].strValue := '';
////TestDummy2_outputparams[4].strKey := '';
////TestDummy2_outputparams[4].strValue := '';
////TestDummy2_outputparams[5].strKey := '';
////TestDummy2_outputparams[5].strValue := '';
////TestDummy2_outputparams[6].strKey := '';
////TestDummy2_outputparams[6].strValue := '';
////TestDummy2_outputparams[7].strKey := '';
////TestDummy2_outputparams[7].strValue := '';
////TestDummy2_outputparams[8].strKey := '';
////TestDummy2_outputparams[8].strValue := '';
////TestDummy2_outputparams[9].strKey := '';
////TestDummy2_outputparams[9].strValue := '';

//M_TestCohapLibrary.init_inpuparams[0].strKey := 'VSupply';
//M_TestCohapLibrary.init_inpuparams[0].strValue := '5.0';
//M_TestCohapLibrary.init_inpuparams[1].strKey := '';
//M_TestCohapLibrary.init_inpuparams[1].strValue := '';
//M_TestCohapLibrary.init_inpuparams[2].strKey := '';
//M_TestCohapLibrary.init_inpuparams[2].strValue := '';

//M_TestCohapLibrary.init_expoutparamlist[0].enumDataType := E_DataType.DT_STRING;
//M_TestCohapLibrary.init_expoutparamlist[0].strVarName := 'returnMsg';
//M_TestCohapLibrary.init_expoutparamlist[1].enumDataType := E_DataType.DT_STRING;
//M_TestCohapLibrary.init_expoutparamlist[1].strVarName := '';
//M_TestCohapLibrary.init_expoutparamlist[2].enumDataType := E_DataType.DT_STRING;
//M_TestCohapLibrary.init_expoutparamlist[2].strVarName := '';

//M_TestCohapLibrary.getSICAndChannelCardVersions_inpuparams[0].strKey := 'channel';
//M_TestCohapLibrary.getSICAndChannelCardVersions_inpuparams[0].strValue := '1';
//M_TestCohapLibrary.getSICAndChannelCardVersions_inpuparams[1].strKey := '';
//M_TestCohapLibrary.getSICAndChannelCardVersions_inpuparams[1].strValue := '';
//M_TestCohapLibrary.getSICAndChannelCardVersions_inpuparams[2].strKey := '';
//M_TestCohapLibrary.getSICAndChannelCardVersions_inpuparams[2].strValue := '';

//M_TestCohapLibrary.getSICAndChannelCardVersions_expoutparamlist[0].enumDataType := E_DataType.DT_STRING;
//M_TestCohapLibrary.getSICAndChannelCardVersions_expoutparamlist[0].strVarName := 'SICVersion';
//M_TestCohapLibrary.getSICAndChannelCardVersions_expoutparamlist[1].enumDataType := E_DataType.DT_STRING;
//M_TestCohapLibrary.getSICAndChannelCardVersions_expoutparamlist[1].strVarName := 'COHAPChannelCardVersion';
//M_TestCohapLibrary.getSICAndChannelCardVersions_expoutparamlist[2].enumDataType := E_DataType.DT_STRING;
//M_TestCohapLibrary.getSICAndChannelCardVersions_expoutparamlist[2].strVarName := '';

//M_TestCohapLibrary.getDLLVersions_inpuparams[0].strKey := '';
//M_TestCohapLibrary.getDLLVersions_inpuparams[0].strValue := '';
//M_TestCohapLibrary.getDLLVersions_inpuparams[1].strKey := '';
//M_TestCohapLibrary.getDLLVersions_inpuparams[1].strValue := '';
//M_TestCohapLibrary.getDLLVersions_inpuparams[2].strKey := '';
//M_TestCohapLibrary.getDLLVersions_inpuparams[2].strValue := '';

//M_TestCohapLibrary.getDLLVersions_expoutparamlist[0].enumDataType := E_DataType.DT_STRING;
//M_TestCohapLibrary.getDLLVersions_expoutparamlist[0].strVarName := 'DUT12133DLLVersion';
//M_TestCohapLibrary.getDLLVersions_expoutparamlist[1].enumDataType := E_DataType.DT_STRING;
//M_TestCohapLibrary.getDLLVersions_expoutparamlist[1].strVarName := 'MUPeT12133DLLVersion';
//M_TestCohapLibrary.getDLLVersions_expoutparamlist[2].enumDataType := E_DataType.DT_STRING;
//M_TestCohapLibrary.getDLLVersions_expoutparamlist[2].strVarName := 'HALDLLVersion';


//M_TestCohapLibrary.initDUT_inpuparams[0].strKey := 'channel';
//M_TestCohapLibrary.initDUT_inpuparams[0].strValue := '1';
//M_TestCohapLibrary.initDUT_inpuparams[1].strKey := 'supplyVoltage';
//M_TestCohapLibrary.initDUT_inpuparams[1].strValue := '5.0';
//M_TestCohapLibrary.initDUT_inpuparams[2].strKey := '';
//M_TestCohapLibrary.initDUT_inpuparams[2].strValue := '';

//M_TestCohapLibrary.initDUT_expoutparamlist[0].enumDataType := E_DataType.DT_STRING;
//M_TestCohapLibrary.initDUT_expoutparamlist[0].strVarName := '';
//M_TestCohapLibrary.initDUT_expoutparamlist[1].enumDataType := E_DataType.DT_STRING;
//M_TestCohapLibrary.initDUT_expoutparamlist[1].strVarName := '';
//M_TestCohapLibrary.initDUT_expoutparamlist[2].enumDataType := E_DataType.DT_STRING;
//M_TestCohapLibrary.initDUT_expoutparamlist[2].strVarName := '';


//M_TestCohapLibrary.readFastChannelData_inputparams[0].strKey := 'channel';
//M_TestCohapLibrary.readFastChannelData_inputparams[0].strValue := '1';
//M_TestCohapLibrary.readFastChannelData_inputparams[1].strKey := '';
//M_TestCohapLibrary.readFastChannelData_inputparams[1].strValue := '';
//M_TestCohapLibrary.readFastChannelData_inputparams[2].strKey := '';
//M_TestCohapLibrary.readFastChannelData_inputparams[2].strValue := '';

//M_TestCohapLibrary.readFastChannelData_expoutparamlist[0].enumDataType := E_DataType.DT_UINT;
//M_TestCohapLibrary.readFastChannelData_expoutparamlist[0].strVarName := 'FastChannel1Data';
//M_TestCohapLibrary.readFastChannelData_expoutparamlist[1].enumDataType := E_DataType.DT_UINT;
//M_TestCohapLibrary.readFastChannelData_expoutparamlist[1].strVarName := 'FastChannel2Data';
//M_TestCohapLibrary.readFastChannelData_expoutparamlist[2].enumDataType := E_DataType.DT_STRING;
//M_TestCohapLibrary.readFastChannelData_expoutparamlist[2].strVarName := 'FastChannel1Status';
//M_TestCohapLibrary.readFastChannelData_expoutparamlist[3].enumDataType := E_DataType.DT_STRING;
//M_TestCohapLibrary.readFastChannelData_expoutparamlist[3].strVarName := 'FastChannel2Status';


//M_TestCohapLibrary.InitLot_inputparams[0].strKey := 'deviceID';
//M_TestCohapLibrary.InitLot_inputparams[0].strValue := '52EMB01-01';
//M_TestCohapLibrary.InitLot_inputparams[1].strKey := 'lotID';
//M_TestCohapLibrary.InitLot_inputparams[1].strValue := '123';
//M_TestCohapLibrary.InitLot_inputparams[2].strKey := 'equipmentID';
//M_TestCohapLibrary.InitLot_inputparams[2].strValue := '1';
//M_TestCohapLibrary.InitLot_inputparams[3].strKey := 'testKind';
//M_TestCohapLibrary.InitLot_inputparams[3].strValue := '1';

//M_TestCohapLibrary.t1Precal_inputparams[0].strKey := 'channel';
//M_TestCohapLibrary.t1Precal_inputparams[0].strValue := '1';
//M_TestCohapLibrary.t1Precal_inputparams[1].strKey := 'deviceID';
//M_TestCohapLibrary.t1Precal_inputparams[1].strValue := '52EMB01-01';
//M_TestCohapLibrary.t1Precal_inputparams[2].strKey := 'temperature';
//M_TestCohapLibrary.t1Precal_inputparams[2].strValue := '-25';
//M_TestCohapLibrary.t1Precal_inputparams[3].strKey := 'force';
//M_TestCohapLibrary.t1Precal_inputparams[3].strValue := '0';
 
//M_TestCohapLibrary.t1Step2_inputparams[0].strKey := 'deviceID';
//M_TestCohapLibrary.t1Step2_inputparams[0].strValue := '52EMB01-01';
//M_TestCohapLibrary.t1Step2_inputparams[1].strKey := 'temperature';
//M_TestCohapLibrary.t1Step2_inputparams[1].strValue := '-25';
//M_TestCohapLibrary.t1Step2_inputparams[2].strKey := 'force';
//M_TestCohapLibrary.t1Step2_inputparams[2].strValue := '40';
 
//M_TestCohapLibrary.t1Step3_inputparams[0].strKey := 'deviceID';
//M_TestCohapLibrary.t1Step3_inputparams[0].strValue := '52EMB01-01';
//M_TestCohapLibrary.t1Step3_inputparams[2].strKey := 'temperature';
//M_TestCohapLibrary.t1Step3_inputparams[2].strValue := '-25';
//M_TestCohapLibrary.t1Step3_inputparams[3].strKey := 'force';
//M_TestCohapLibrary.t1Step3_inputparams[3].strValue := '0';



{------------------------}
strDeviceName := 'Device12133';

readSerialNumber_inpuparams[0].strKey := 'channel';
readSerialNumber_inpuparams[0].strValue := '1';
readSerialNumber_inpuparams[1].strKey := '';
readSerialNumber_inpuparams[1].strValue := '';
readSerialNumber_inpuparams[2].strKey := '';
readSerialNumber_inpuparams[2].strValue := '';

readSerialNumber_expoutparamlist[0].enumDataType := E_DataType.DT_ULINT;
readSerialNumber_expoutparamlist[0].strVarName := 'serialnumber';
readSerialNumber_expoutparamlist[1].enumDataType := E_DataType.DT_STRING;
readSerialNumber_expoutparamlist[1].strVarName := 'stringserialno';
readSerialNumber_expoutparamlist[2].enumDataType := E_DataType.DT_STRING;
readSerialNumber_expoutparamlist[2].strVarName := '';


ReadDeviceOutput_inpuparams[0].strKey := 'channel';
ReadDeviceOutput_inpuparams[0].strValue := '1';
ReadDeviceOutput_inpuparams[1].strKey := '';
ReadDeviceOutput_inpuparams[1].strValue := '';
ReadDeviceOutput_inpuparams[2].strKey := '';
ReadDeviceOutput_inpuparams[2].strValue := '';

ReadDeviceOutput_expoutparamlist[0].enumDataType := E_DataType.DT_INT;
ReadDeviceOutput_expoutparamlist[0].strVarName := 'P1data';
ReadDeviceOutput_expoutparamlist[1].enumDataType := E_DataType.DT_INT;
ReadDeviceOutput_expoutparamlist[1].strVarName := 'P1out';
ReadDeviceOutput_expoutparamlist[2].enumDataType := E_DataType.DT_INT;
ReadDeviceOutput_expoutparamlist[2].strVarName := 'P2data';
ReadDeviceOutput_expoutparamlist[3].enumDataType := E_DataType.DT_INT;
ReadDeviceOutput_expoutparamlist[3].strVarName := 'P2out';
ReadDeviceOutput_expoutparamlist[4].enumDataType := E_DataType.DT_INT;
ReadDeviceOutput_expoutparamlist[4].strVarName := 'T1data';
ReadDeviceOutput_expoutparamlist[5].enumDataType := E_DataType.DT_INT;
ReadDeviceOutput_expoutparamlist[5].strVarName := 'T1out';
ReadDeviceOutput_expoutparamlist[6].enumDataType := E_DataType.DT_INT;
ReadDeviceOutput_expoutparamlist[6].strVarName := 'T2data';
ReadDeviceOutput_expoutparamlist[7].enumDataType := E_DataType.DT_INT;
ReadDeviceOutput_expoutparamlist[7].strVarName := 'T2out';

PowerUp_inpuparams[0].strKey := 'channel';
PowerUp_inpuparams[0].strValue := '1';
PowerUp_inpuparams[1].strKey := 'supplyVoltage';
PowerUp_inpuparams[1].strValue := '5.0';
PowerUp_inpuparams[2].strKey := '';
PowerUp_inpuparams[2].strValue := '';

PowerUp_expoutparamlist[0].enumDataType := E_DataType.DT_DOUBLE;
PowerUp_expoutparamlist[0].strVarName := 'Vsupply';
PowerUp_expoutparamlist[1].enumDataType := E_DataType.DT_DOUBLE;
PowerUp_expoutparamlist[1].strVarName := 'current';
PowerUp_expoutparamlist[2].enumDataType := E_DataType.DT_STRING;
PowerUp_expoutparamlist[2].strVarName := '';

PowerDown_inpuparams[0].strKey := 'channel';
PowerDown_inpuparams[0].strValue := '1';
PowerDown_inpuparams[1].strKey := '';
PowerDown_inpuparams[1].strValue := '';
PowerDown_inpuparams[2].strKey := '';
PowerDown_inpuparams[2].strValue := '';

PowerDown_expoutparamlist[0].enumDataType := E_DataType.DT_STRING;
PowerDown_expoutparamlist[0].strVarName := '';
PowerDown_expoutparamlist[1].enumDataType := E_DataType.DT_STRING;
PowerDown_expoutparamlist[1].strVarName := '';
PowerDown_expoutparamlist[2].enumDataType := E_DataType.DT_STRING;
PowerDown_expoutparamlist[2].strVarName := '';

TestDummy_inpuparams[0].strKey := 'channel';
TestDummy_inpuparams[0].strValue := '1';
TestDummy_inpuparams[1].strKey := 'bInput';
TestDummy_inpuparams[1].strValue := 'FALSE';
TestDummy_inpuparams[2].strKey := '';
TestDummy_inpuparams[2].strValue := '';

TestDummy_expoutparamlist[0].enumDataType := E_DataType.DT_STRING;
TestDummy_expoutparamlist[0].strVarName := 'serialno';
TestDummy_expoutparamlist[1].enumDataType := E_DataType.DT_DOUBLE;
TestDummy_expoutparamlist[1].strVarName := 'Voltage';
TestDummy_expoutparamlist[2].enumDataType := E_DataType.DT_BOOL;
TestDummy_expoutparamlist[2].strVarName := 'MethodResponse';
TestDummy_expoutparamlist[3].enumDataType := E_DataType.DT_UINT;
TestDummy_expoutparamlist[3].strVarName := 'current';
TestDummy_expoutparamlist[4].enumDataType := E_DataType.DT_STRING;
TestDummy_expoutparamlist[4].strVarName := 'P1status';
TestDummy_expoutparamlist[5].enumDataType := E_DataType.DT_STRING;
TestDummy_expoutparamlist[5].strVarName := 'P2status';

TestDummy2_inpuparams[0].strKey := 'channel';
TestDummy2_inpuparams[0].strValue := '1';
TestDummy2_inpuparams[1].strKey := 'Input2';
TestDummy2_inpuparams[1].strValue := 'dummyimput2';
TestDummy2_inpuparams[2].strKey := '';
TestDummy2_inpuparams[2].strValue := '';

TestDummy2_expoutparamlist[0].enumDataType := E_DataType.DT_INT;
TestDummy2_expoutparamlist[0].strVarName := 'output1';
TestDummy2_expoutparamlist[1].enumDataType := E_DataType.DT_STRING;
TestDummy2_expoutparamlist[1].strVarName := 'output2';
TestDummy2_expoutparamlist[2].enumDataType := E_DataType.DT_ULINT;
TestDummy2_expoutparamlist[2].strVarName := 'fastchannel1';
TestDummy2_expoutparamlist[3].enumDataType := E_DataType.DT_ULINT;
TestDummy2_expoutparamlist[3].strVarName := 'fastchannel2';
TestDummy2_expoutparamlist[4].enumDataType := E_DataType.DT_STRING;
TestDummy2_expoutparamlist[4].strVarName := 'fastchannel3';
TestDummy2_expoutparamlist[5].enumDataType := E_DataType.DT_INT;
TestDummy2_expoutparamlist[5].strVarName := 'fastchannel4';
TestDummy2_expoutparamlist[6].enumDataType := E_DataType.DT_ULINT;
TestDummy2_expoutparamlist[6].strVarName := 'fastchannel5';
TestDummy2_expoutparamlist[7].enumDataType := E_DataType.DT_ULINT;
TestDummy2_expoutparamlist[7].strVarName := 'fastchannel6';
TestDummy2_expoutparamlist[8].enumDataType := E_DataType.DT_STRING;
TestDummy2_expoutparamlist[8].strVarName := 'fastchannel7';
TestDummy2_expoutparamlist[9].enumDataType := E_DataType.DT_INT;
TestDummy2_expoutparamlist[9].strVarName := 'fastchannel8';

//TestDummy2_outputparams[0].strKey := '';
//TestDummy2_outputparams[0].strValue := '';
//TestDummy2_outputparams[1].strKey := '';
//TestDummy2_outputparams[1].strValue := '';
//TestDummy2_outputparams[2].strKey := '';
//TestDummy2_outputparams[2].strValue := '';
//TestDummy2_outputparams[3].strKey := '';
//TestDummy2_outputparams[3].strValue := '';
//TestDummy2_outputparams[4].strKey := '';
//TestDummy2_outputparams[4].strValue := '';
//TestDummy2_outputparams[5].strKey := '';
//TestDummy2_outputparams[5].strValue := '';
//TestDummy2_outputparams[6].strKey := '';
//TestDummy2_outputparams[6].strValue := '';
//TestDummy2_outputparams[7].strKey := '';
//TestDummy2_outputparams[7].strValue := '';
//TestDummy2_outputparams[8].strKey := '';
//TestDummy2_outputparams[8].strValue := '';
//TestDummy2_outputparams[9].strKey := '';
//TestDummy2_outputparams[9].strValue := '';

init_inpuparams[0].strKey := 'VSupply';
init_inpuparams[0].strValue := '5.0';
init_inpuparams[1].strKey := '';
init_inpuparams[1].strValue := '';
init_inpuparams[2].strKey := '';
init_inpuparams[2].strValue := '';

init_expoutparamlist[0].enumDataType := E_DataType.DT_STRING;
init_expoutparamlist[0].strVarName := 'returnMsg';
init_expoutparamlist[1].enumDataType := E_DataType.DT_STRING;
init_expoutparamlist[1].strVarName := '';
init_expoutparamlist[2].enumDataType := E_DataType.DT_STRING;
init_expoutparamlist[2].strVarName := '';

getSICAndChannelCardVersions_inpuparams[0].strKey := 'channel';
getSICAndChannelCardVersions_inpuparams[0].strValue := '1';
getSICAndChannelCardVersions_inpuparams[1].strKey := '';
getSICAndChannelCardVersions_inpuparams[1].strValue := '';
getSICAndChannelCardVersions_inpuparams[2].strKey := '';
getSICAndChannelCardVersions_inpuparams[2].strValue := '';

getSICAndChannelCardVersions_expoutparamlist[0].enumDataType := E_DataType.DT_STRING;
getSICAndChannelCardVersions_expoutparamlist[0].strVarName := 'SICVersion';
getSICAndChannelCardVersions_expoutparamlist[1].enumDataType := E_DataType.DT_STRING;
getSICAndChannelCardVersions_expoutparamlist[1].strVarName := 'COHAPChannelCardVersion';
getSICAndChannelCardVersions_expoutparamlist[2].enumDataType := E_DataType.DT_STRING;
getSICAndChannelCardVersions_expoutparamlist[2].strVarName := '';

getDLLVersions_inpuparams[0].strKey := '';
getDLLVersions_inpuparams[0].strValue := '';
getDLLVersions_inpuparams[1].strKey := '';
getDLLVersions_inpuparams[1].strValue := '';
getDLLVersions_inpuparams[2].strKey := '';
getDLLVersions_inpuparams[2].strValue := '';

getDLLVersions_expoutparamlist[0].enumDataType := E_DataType.DT_STRING;
getDLLVersions_expoutparamlist[0].strVarName := 'DUT12133DLLVersion';
getDLLVersions_expoutparamlist[1].enumDataType := E_DataType.DT_STRING;
getDLLVersions_expoutparamlist[1].strVarName := 'MUPeT12133DLLVersion';
getDLLVersions_expoutparamlist[2].enumDataType := E_DataType.DT_STRING;
getDLLVersions_expoutparamlist[2].strVarName := 'HALDLLVersion';


initDUT_inpuparams[0].strKey := 'channel';
initDUT_inpuparams[0].strValue := '1';
initDUT_inpuparams[1].strKey := 'supplyVoltage';
initDUT_inpuparams[1].strValue := '5.0';
initDUT_inpuparams[2].strKey := '';
initDUT_inpuparams[2].strValue := '';

initDUT_expoutparamlist[0].enumDataType := E_DataType.DT_STRING;
initDUT_expoutparamlist[0].strVarName := '';
initDUT_expoutparamlist[1].enumDataType := E_DataType.DT_STRING;
initDUT_expoutparamlist[1].strVarName := '';
initDUT_expoutparamlist[2].enumDataType := E_DataType.DT_STRING;
initDUT_expoutparamlist[2].strVarName := '';


readFastChannelData_inputparams[0].strKey := 'channel';
readFastChannelData_inputparams[0].strValue := '1';
readFastChannelData_inputparams[1].strKey := '';
readFastChannelData_inputparams[1].strValue := '';
readFastChannelData_inputparams[2].strKey := '';
readFastChannelData_inputparams[2].strValue := '';

readFastChannelData_expoutparamlist[0].enumDataType := E_DataType.DT_UINT;
readFastChannelData_expoutparamlist[0].strVarName := 'FastChannel1Data';
readFastChannelData_expoutparamlist[1].enumDataType := E_DataType.DT_UINT;
readFastChannelData_expoutparamlist[1].strVarName := 'FastChannel2Data';
readFastChannelData_expoutparamlist[2].enumDataType := E_DataType.DT_STRING;
readFastChannelData_expoutparamlist[2].strVarName := 'FastChannel1Status';
readFastChannelData_expoutparamlist[3].enumDataType := E_DataType.DT_STRING;
readFastChannelData_expoutparamlist[3].strVarName := 'FastChannel2Status';


InitLot_inputparams[0].strKey := 'deviceID';
InitLot_inputparams[0].strValue := '52EMB01-01';
InitLot_inputparams[1].strKey := 'lotID';
InitLot_inputparams[1].strValue := '123';
InitLot_inputparams[2].strKey := 'equipmentID';
InitLot_inputparams[2].strValue := '1';
InitLot_inputparams[3].strKey := 'testKind';
InitLot_inputparams[3].strValue := '1';

t1Precal_inputparams[0].strKey := 'channel';
t1Precal_inputparams[0].strValue := '1';
t1Precal_inputparams[1].strKey := 'deviceID';
t1Precal_inputparams[1].strValue := '52EMB01-01';
t1Precal_inputparams[2].strKey := 'temperature';
t1Precal_inputparams[2].strValue := '-25';
t1Precal_inputparams[3].strKey := 'force';
t1Precal_inputparams[3].strValue := '0';
 
t1Step2_inputparams[0].strKey := 'deviceID';
t1Step2_inputparams[0].strValue := '52EMB01-01';
t1Step2_inputparams[1].strKey := 'temperature';
t1Step2_inputparams[1].strValue := '-25';
t1Step2_inputparams[2].strKey := 'force';
t1Step2_inputparams[2].strValue := '40';
 
t1Step3_inputparams[0].strKey := 'deviceID';
t1Step3_inputparams[0].strValue := '52EMB01-01';
t1Step3_inputparams[2].strKey := 'temperature';
t1Step3_inputparams[2].strValue := '-25';
t1Step3_inputparams[3].strKey := 'force';
t1Step3_inputparams[3].strValue := '0';
END_ACTION

ACTION A_LaserMarkingParams:
IF bConnectToLaserMarker THEN
	bRes_LaserConnected := MyLaser1.M_Connect();
	IF bRes_LaserConnected THEN
	//Add some timer based logic to do error handling.
		bConnectToLaserMarker := FALSE;
	ELSIF MyLaser1.P_bError THEN
		bConnectToLaserMarker := FALSE;
		MyLaser1.M_ClearError();
	END_IF
END_IF


IF bDisconnectFromLaserMarker THEN
	bRes_LaserDisconnected := MyLaser1.M_Disconnect();
	IF bRes_LaserDisconnected THEN
		bDisconnectFromLaserMarker := FALSE;
	ELSIF MyLaser1.P_bError THEN
		bDisconnectFromLaserMarker := FALSE;
		MyLaser1.M_ClearError();
	END_IF
END_IF


IF bPeakCurrentProgramInLaser THEN
	bRes_PeakCurrentProgramInLaser := MyLaser1.M_PeakCurrentProgram();
	IF bRes_PeakCurrentProgramInLaser THEN
		bPeakCurrentProgramInLaser := FALSE;
	ELSIF MyLaser1.P_bError THEN
		bPeakCurrentProgramInLaser := FALSE;
		MyLaser1.M_ClearError();
	END_IF
END_IF


IF bSendProgramToLaser THEN
	bRes_SendProgramtoLaser := MyLaser1.M_SendProgramtoLaser(filepath,LaserMemoryLocation);
	IF bRes_SendProgramtoLaser THEN
		bSendProgramToLaser := FALSE;
	ELSIF MyLaser1.P_bError THEN
		bSendProgramToLaser := FALSE;
		MyLaser1.M_ClearError();
	END_IF
END_IF

IF bSaveCurrentLaserProgramtoPC THEN
	bRes_SaveCurrentLaserProgramtoPC := MyLaser1.M_SaveCurrentLaserProgramtoPC(LaserProgramFolderPath, out_bool_SaveProgramToPC_Success => SaveCurrentLaserProgramToPCSuccess);
	IF bRes_SaveCurrentLaserProgramtoPC THEN
//		SaveCurrentLaserProgramToPCSuccess := MyLaser1
		bSaveCurrentLaserProgramtoPC := FALSE;
	ELSIF MyLaser1.P_bError THEN
		bSaveCurrentLaserProgramtoPC := FALSE;
		MyLaser1.M_ClearError();
	END_IF
END_IF

IF bGetCurrentProgram THEN
	bRes_GetCurrentProgram := MyLaser1.M_GetCurrentProgram(strCurrentProgram => CurrentProgramName);
	IF bRes_GetCurrentProgram THEN
		bGetCurrentProgram := FALSE;
	ELSIF MyLaser1.P_bError THEN
		bGetCurrentProgram := FALSE;
		MyLaser1.M_ClearError();
	END_IF
END_IF

IF bStartMarking THEN
	bRes_StartMarking := MyLaser1.M_StartMarking();
	IF bRes_StartMarking THEN
		bStartMarking := FALSE;
	ELSIF MyLaser1.P_bError THEN
		bStartMarking := FALSE;
		MyLaser1.M_ClearError();
	END_IF
END_IF

IF bStopMarking THEN
	bRes_StopMarking := MyLaser1.M_StopMarking();
	IF bRes_StopMarking THEN
		bStopMarking := FALSE;
	ELSIF MyLaser1.P_bError THEN
		bStopMarking := FALSE;
		MyLaser1.M_ClearError();
	END_IF
END_IF

IF bResetErrors THEN
	bRes_Reset := MyLaser1.M_Reset();
	IF bRes_Reset THEN
		bResetErrors := FALSE;
	ELSIF MyLaser1.P_bError THEN
		bResetErrors := FALSE;
		MyLaser1.M_ClearError();
	END_IF
END_IF

//IF bUpdateProgramBlockInTheLaser THEN
//	bRes_UpdateProgramBlockInTheLaser := MyLaser1.M_UpdateSingleProgramBlockData(LaserMemoryLocation, _blockNumber, _blockData, _blockType, out_bool_UpdateData_Success => _bUpdateSingleBlockDataSuccess);
//	IF bRes_UpdateProgramBlockInTheLaser THEN
//		bUpdateProgramBlockInTheLaser := FALSE;
//	ELSIF MyLaser1.P_bError THEN
//		bUpdateProgramBlockInTheLaser := FALSE;
//		MyLaser1.M_ClearError();
//	END_IF
//END_IF

IF bUpdateProgramBlockInTheLaser THEN
	bRes_UpdateProgramBlockInTheLaser := MyLaser1.M_UpdateSingleBlockMarkingInformation(_blockNumber, _blockData, _bool_markenabled);
	IF bRes_UpdateProgramBlockInTheLaser THEN
		bUpdateProgramBlockInTheLaser := FALSE;
	ELSIF MyLaser1.P_bError THEN
		bUpdateProgramBlockInTheLaser := FALSE;
		MyLaser1.M_ClearError();
	END_IF
END_IF

IF bUpdateProgramBlockMarkEnabledInTheLaser THEN
	bRes_UpdateProgramBlockMarkEnabledInTheLaser := MyLaser1.M_UpdateSingleProgramBlockMarkEnabled( LaserProgramMemoryLocation := LaserMemoryLocation, BlockNumber := _blockNumber, BlockType := _blockType ,MarkEnabled := _bool_markenabled ,out_bool_MarkEnabled_Success => _bUpdateSingleBlockMarkEnabled_Success);
	IF bRes_UpdateProgramBlockMarkEnabledInTheLaser THEN
		bUpdateProgramBlockMarkEnabledInTheLaser := FALSE;
	ELSIF MyLaser1.P_bError THEN
		bUpdateProgramBlockMarkEnabledInTheLaser := FALSE;
		MyLaser1.M_ClearError();
	END_IF
END_IF

IF bGetLaserStatus THEN
	bRes_GetLaserStatus := MyLaser1.M_GetLaserStatus( out_string_laserStatus => _string_laserstatus);
	IF bRes_GetLaserStatus THEN
		bGetLaserStatus := FALSE;
	ELSIF MyLaser1.P_bError THEN
		bGetLaserStatus := FALSE;
		MyLaser1.M_ClearError();
	END_IF
END_IF

IF bGetLaserErrorStatus THEN
	bRes_GetLaserErrorStatus := MyLaser1.M_GetLaserErrorStatus( out_bool_IsLaserError => _bIsLaserError);
	IF bRes_GetLaserErrorStatus THEN
		bGetLaserErrorStatus := FALSE;
	ELSIF MyLaser1.P_bError THEN
		bGetLaserErrorStatus := FALSE;
		MyLaser1.M_ClearError();
	END_IF
END_IF

IF bGetLaserActivatedStatus THEN
	bRes_GetLaserActivatedStatus := MyLaser1.M_GetLaserActivatedStatus( out_IsLaserActivated => _bIsLaserActivated);
	IF bRes_GetLaserActivatedStatus THEN
		bGetLaserActivatedStatus := FALSE;
	ELSIF MyLaser1.P_bError THEN
		bGetLaserActivatedStatus := FALSE;
		MyLaser1.M_ClearError();
	END_IF
END_IF

IF bGetLaserMarkingStatus THEN
	bRes_GetLaserMarkingStatus := MyLaser1.M_GetLaserMarkingStatus( out_bool_IsLaserMarking => _bIsLaserMarking);
	IF bRes_GetLaserMarkingStatus THEN
		bGetLaserMarkingStatus := FALSE;
	ELSIF MyLaser1.P_bError THEN
		bGetLaserMarkingStatus := FALSE;
		MyLaser1.M_ClearError();
	END_IF
END_IF

IF _OneTimeArrayBuild THEN
	FOR intIndex2 := 0 TO 255 DO
		IF intIndex2 <= LastBlockToMark THEN
			BlockInfoArray[intIndex2].MarkEnabled := TRUE;
			_tempString := CONCAT('Block', INT_TO_STRING(intIndex2));
			BlockInfoArray[intIndex2].BlockText := _tempString;
		ELSE
			BlockInfoArray[intIndex2].MarkEnabled := FALSE;	
			BlockInfoArray[intIndex2].BlockText := '';
		END_IF
	END_FOR
	_OneTimeArrayBuild := FALSE;
END_IF

IF bUpdateAllMarkingInfo_MethodCall THEN
	bRes_UpdateAllMarkingInfo_MethodCall := MyLaser1.M_UpdateAllMarkingInformation(LastBlockToMark);
	bUpdateAllMarkingInfo_MethodCall := FALSE;
END_IF
IF MyLaser1.P_bError THEN
	bUpdateAllMarkingInfo_MethodCall := FALSE;
	MyLaser1.M_ClearError();
END_IF

IF bUpdateAllMarkingInfo THEN
	CASE inst_intStep OF
		0: //Check for errors and Integer value which we are gonna run the update single block information
				IF MyLaser1.P_bError THEN
					inst_intStep := 0;
					bUpdateAllMarkingInfo := FALSE;
				ELSE
					inst_intStep := 10;
				END_IF
		10: // Run the M_UpdateSingleBlockMarkingInformation Command
				bRes_UpdateAllMarkInfo[intIndex] := MyLaser1.M_UpdateSingleBlockMarkingInformation(intIndex ,BlockInfoArray[intIndex].BlockText, BlockInfoArray[intIndex].MarkEnabled);
				IF bRes_UpdateAllMarkInfo[intIndex] THEN 
					inst_intStep := 20;
				ELSIF MyLaser1.P_bError THEN
					inst_intStep := 0;
					intIndex :=0;
					bUpdateAllMarkingInfo := FALSE;
				END_IF
		20: // Check if the M_UpdateSingleBlockMarkingInformation command failed or passed
				IF bRes_UpdateAllMarkInfo[LastBlockToMark] OR NOT bRes_UpdateAllMarkInfo[intIndex] OR (intIndex = LastBlockToMark) THEN //This means we reached the final element update
					bUpdateAllMarkingInfo := FALSE;
					intIndex :=0;
					inst_intStep := 0;
				ELSIF bRes_UpdateAllMarkInfo[intIndex] THEN
					inst_intStep := 0;
					intIndex := intIndex + 1;
				ELSIF MyLaser1.P_bError THEN
					bUpdateAllMarkingInfo := FALSE;
					MyLaser1.M_ClearError();	
				END_IF			
	END_CASE
END_IF

IF bGetLimitsFromDB THEN
	_inst_bDataTransferred := fbDataHandler.M_TransferData(in_strParametersDatabaseName);
	IF _inst_bDataTransferred THEN
		bGetLimitsFromDB := FALSE;
	ELSIF fbDataHandler.P_bError THEN
		bGetLimitsFromDB := FALSE;
		fbDataHandler.M_ClearError();
	END_IF
END_IF

IF bGetLaserParamsFromDB_L1 THEN
	_inst_bLaserLimitsDataTransferred_L1 := fbDataHandler.M_TransferData(in_strParametersDBNameLaserLimits_L1);
	IF _inst_bLaserLimitsDataTransferred_L1 THEN
		bGetLaserParamsFromDB_L1 := FALSE;
		ELSIF fbDataHandler.P_bError THEN
			bGetLaserParamsFromDB_L1 := FALSE;
			fbDataHandler.M_ClearError();
	END_IF
END_IF

IF bGetLaserParamsFromDB_L2 THEN
	_inst_bLaserLimitsDataTransferred_L2 := fbDataHandler.M_TransferData(in_strParametersDBNameLaserLimits_L2);
	IF _inst_bLaserLimitsDataTransferred_L2 THEN
		bGetLaserParamsFromDB_L2 := FALSE;
		ELSIF fbDataHandler.P_bError THEN
			bGetLaserParamsFromDB_L2 := FALSE;
			fbDataHandler.M_ClearError();
	END_IF
END_IF

IF bGetLaserParamsFromDB_R1 THEN
	_inst_bLaserLimitsDataTransferred_R1 := fbDataHandler.M_TransferData(in_strParametersDBNameLaserLimits_R1);
	IF _inst_bLaserLimitsDataTransferred_R1 THEN
		bGetLaserParamsFromDB_R1 := FALSE;
		ELSIF fbDataHandler.P_bError THEN
			bGetLaserParamsFromDB_R1 := FALSE;
			fbDataHandler.M_ClearError();
	END_IF
END_IF

IF bGetLaserParamsFromDB_R2 THEN
	_inst_bLaserLimitsDataTransferred_R2 := fbDataHandler.M_TransferData(in_strParametersDBNameLaserLimits_R2);
	IF _inst_bLaserLimitsDataTransferred_R2 THEN
		bGetLaserParamsFromDB_R2 := FALSE;
		ELSIF fbDataHandler.P_bError THEN
			bGetLaserParamsFromDB_R2 := FALSE;
			fbDataHandler.M_ClearError();
	END_IF
END_IF

IF bPerformPriorOp_Smart THEN
	_inst_bPriorOp_Smart := fbDataHandler2.M_TransferData(in_strParametersDBName_SmartWater);
	IF _inst_bPriorOp_Smart THEN
		bPerformPriorOp_Smart := FALSE;
	ELSIF fbDataHandler2.P_bError THEN 
		bPerformPriorOp_Smart := FALSE;
		fbDataHandler2.M_ClearError();
	END_IF
END_IF

IF bPerformPriorOp_FFT THEN
	_inst_bPriorOp_FFT := fbDataHandler.M_TransferData(in_strParametersDBName_FFTLaser_L1);
	IF _inst_bPriorOp_FFT THEN
		bPerformPriorOp_FFT := FALSE;
	ELSIF fbDataHandler.P_bError THEN 
		bPerformPriorOp_FFT := FALSE;
		fbDataHandler.M_ClearError();
	END_IF
END_IF

Temp_CR_LOOKUP_NestL1 := FIND('GV354-006:220705-141019_CR','_CR');
iLengthDataMatrixNestL1 := LEN('GV354-006:220705-141019_CR');
IF  (Temp_CR_LOOKUP_NestL1 > 0) THEN
	ParamsArrayNestA := REPLACE('GV354-006:220705-141019_CR', concat(' CR ' , '0.023456'),6,iLengthDataMatrixNestL1 - 2);
END_IF
END_ACTION

ACTION A_Machine:
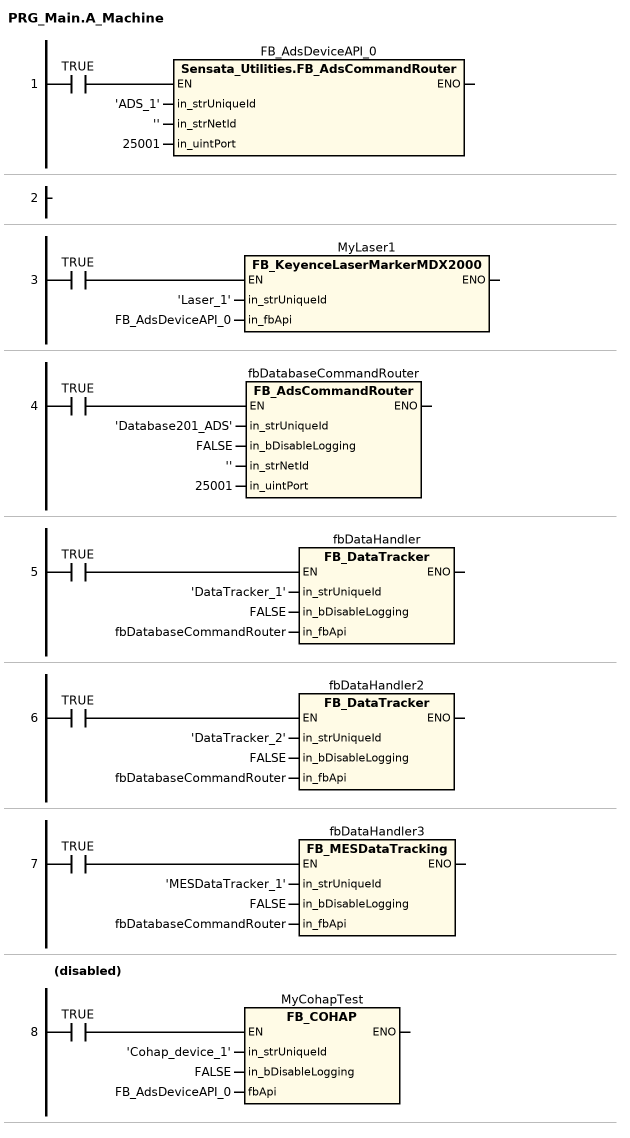
// NETWORK 1
FB_AdsDeviceAPI_0(in_strUniqueId := 'ADS_1', in_strNetId := '', in_uintPort := 25001); // Sensata_Utilities.FB_AdsCommandRouter

// NETWORK 2

// NETWORK 3
MyLaser1(in_strUniqueId := 'Laser_1', in_fbApi := FB_AdsDeviceAPI_0); // FB_KeyenceLaserMarkerMDX2000

// NETWORK 4
fbDatabaseCommandRouter(
    in_strUniqueId := 'Database201_ADS',
    in_bDisableLogging := FALSE,
    in_strNetId := '',
    in_uintPort := 25001); // FB_AdsCommandRouter

// NETWORK 5
fbDataHandler(
    in_strUniqueId := 'DataTracker_1',
    in_bDisableLogging := FALSE,
    in_fbApi := fbDatabaseCommandRouter); // FB_DataTracker

// NETWORK 6
fbDataHandler2(
    in_strUniqueId := 'DataTracker_2',
    in_bDisableLogging := FALSE,
    in_fbApi := fbDatabaseCommandRouter); // FB_DataTracker

// NETWORK 7
fbDataHandler3(
    in_strUniqueId := 'MESDataTracker_1',
    in_bDisableLogging := FALSE,
    in_fbApi := fbDatabaseCommandRouter); // FB_MESDataTracking

// NETWORK 8 (disabled)
// MyCohapTest(in_strUniqueId := 'Cohap_device_1', in_bDisableLogging := FALSE, fbApi := FB_AdsDeviceAPI_0); // FB_COHAP
END_ACTION

ACTION A_MESVars:

IF bPerformGetLotInfoFromLotBarcode THEN
	_inst_bGetLotInfo_LotBarcode := fbDataHandler3.M_TransferData(in_strParamDBName_GetLotInfo);
	IF _inst_bGetLotInfo_LotBarcode THEN
		bPerformGetLotInfoFromLotBarcode := FALSE;
	ELSIF fbDataHandler3.P_bError THEN 
		bPerformGetLotInfoFromLotBarcode := FALSE;
		fbDataHandler3.M_ClearError();
	END_IF
END_IF

IF bPerformGetOpInfoFromOpBarcode THEN
	_inst_bGetOpInfo_OpBarcode := fbDataHandler3.M_TransferData(in_strParamDBName_GetOpInfo);
	IF _inst_bGetOpInfo_OpBarcode THEN
		bPerformGetOpInfoFromOpBarcode := FALSE;
	ELSIF fbDataHandler3.P_bError THEN 
		bPerformGetOpInfoFromOpBarcode := FALSE;
		fbDataHandler3.M_ClearError();
	END_IF
END_IF

IF bPerformStartLot THEN
	_inst_bStartLot := fbDataHandler3.M_TransferData(in_strParamDBName_StartLot);
	IF _inst_bStartLot THEN
		bPerformStartLot := FALSE;
	ELSIF fbDataHandler3.P_bError THEN 
		bPerformStartLot := FALSE;
		fbDataHandler3.M_ClearError();
	END_IF
END_IF

IF bPerformGetProdLotComponents THEN
	_inst_bGetProdLotComponents := fbDataHandler3.M_TransferData(in_strParamDBName_GetProdLotComps);
	IF _inst_bGetProdLotComponents THEN
		bPerformGetProdLotComponents := FALSE;
	ELSIF fbDataHandler3.P_bError THEN 
		bPerformGetProdLotComponents := FALSE;
		fbDataHandler3.M_ClearError();
	END_IF
END_IF


IF bPerformComponentValidation1 THEN
	_inst_bCompValidation1 := fbDataHandler3.M_TransferData(in_strParamDBName_Comp1Validation1);
	IF _inst_bCompValidation1 THEN
		bPerformComponentValidation1 := FALSE;
	ELSIF fbDataHandler3.P_bError THEN 
		bPerformComponentValidation1 := FALSE;
		fbDataHandler3.M_ClearError();
	END_IF
END_IF

IF bPerformComponentValidation2 THEN
	_inst_bCompValidation2 := fbDataHandler3.M_TransferData(in_strParamDBName_Comp1Validation2);
	IF _inst_bCompValidation2 THEN
		bPerformComponentValidation2 := FALSE;
	ELSIF fbDataHandler3.P_bError THEN 
		bPerformComponentValidation2 := FALSE;
		fbDataHandler3.M_ClearError();
	END_IF
END_IF

IF bPerformComponentValidation3 THEN
	_inst_bCompValidation3 := fbDataHandler3.M_TransferData(in_strParamDBName_Comp1Validation3);
	IF _inst_bCompValidation3 THEN
		bPerformComponentValidation3 := FALSE;
	ELSIF fbDataHandler3.P_bError THEN 
		bPerformComponentValidation3 := FALSE;
		fbDataHandler3.M_ClearError();
	END_IF
END_IF

IF bPerformGetMachineSettings THEN
	_inst_bGetMachineSettings := fbDataHandler3.M_TransferData(in_strParamDBName_GetMachSetting);
	IF _inst_bGetMachineSettings THEN
		bPerformGetMachineSettings := FALSE;
	ELSIF fbDataHandler3.P_bError THEN 
		bPerformGetMachineSettings := FALSE;
		fbDataHandler3.M_ClearError();
	END_IF
END_IF

IF bPerformAddScrapCompByReason THEN
	_inst_bAddScrapCompByReason := fbDataHandler3.M_TransferData(in_strParamDBName_AddScrapCompByReason);
	IF _inst_bAddScrapCompByReason THEN
		bPerformAddScrapCompByReason := FALSE;
	ELSIF fbDataHandler3.P_bError THEN 
		bPerformAddScrapCompByReason := FALSE;
		fbDataHandler3.M_ClearError();
	END_IF
END_IF

IF bPerformEndLotComp THEN
	_inst_bEndLotComp := fbDataHandler3.M_TransferData(in_strParamDBName_EndLotComp);
	IF _inst_bEndLotComp THEN
		bPerformEndLotComp := FALSE;
	ELSIF fbDataHandler3.P_bError THEN 
		bPerformEndLotComp := FALSE;
		fbDataHandler3.M_ClearError();
	END_IF
END_IF

IF bPerformGetMachineDefects THEN
	_inst_bGetMachineDefects := fbDataHandler3.M_TransferData(in_strParamDBName_GetMachDefects);
	IF _inst_bGetMachineDefects THEN
		bPerformGetMachineDefects := FALSE;
	ELSIF fbDataHandler3.P_bError THEN 
		bPerformGetMachineDefects := FALSE;
		fbDataHandler3.M_ClearError();
	END_IF
END_IF
END_ACTION

ACTION A_Station1:
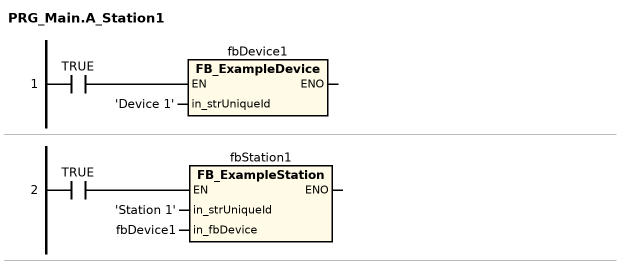
// NETWORK 1
fbDevice1(in_strUniqueId := 'Device 1'); // FB_ExampleDevice

// NETWORK 2
fbStation1(in_strUniqueId := 'Station 1', in_fbDevice := fbDevice1); // FB_ExampleStation
END_ACTION

ACTION A_Station2:
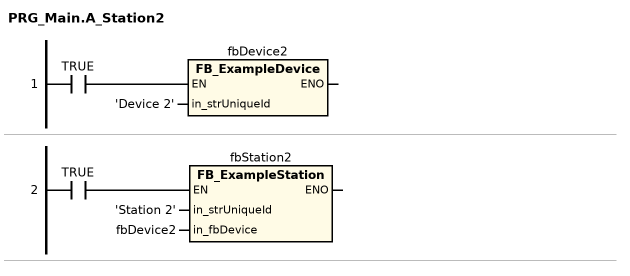
// NETWORK 1
fbDevice2(in_strUniqueId := 'Device 2'); // FB_ExampleDevice

